(* IEC 61131-3 sources: scada_scout/plc_programs (part 4) *)

(* ---- PRG_GPS02LBB01.st ---- *)
(* ========================================================================
   PLC PROGRAM: PRG_GPS02LBB01
   IED: GPS02LBB01
   Device: GPS02LBB01
   Generated: 2026-02-05 10:51:36

   This program runs cyclically (default 100ms) and has access to all
   data points of the associated IEC 61850 device. Users can add custom
   logic in the designated sections below.
   ======================================================================== *)

PROGRAM PRG_GPS02LBB01
VAR
    (* ====== System Variables ====== *)
    cycle_count: UDINT := 0;           (* Increments each scan cycle *)
    first_scan: BOOL := TRUE;          (* TRUE only on first execution *)
    scan_time_ms: REAL := 0.0;         (* Last scan time in milliseconds *)

    (* ====== IED Connection Status ====== *)
    ied_connected: BOOL := FALSE;      (* TRUE when IED server is running *)
    ied_name: STRING := 'GPS02LBB01';
    device_name: STRING := 'GPS02LBB01';

    (* ====== Logical Devices ====== *)
    (* Available LDs: AnUn_ArcProtInput1, Application, BinIO, BinIO_BinaryInputs, BinIO_BinaryOutputs, CB1, CB1_Fundamental, Ds1, Ds2, Mod1, Mod1_Channel1, Mod2, Mod2_Channel1, Mod3, Mod3_Channel1, PowS, PowS_MeasPointI3ph1, PowS_MeasPointV3ph1, Rec, Rec_FaultRecorder, VI3p1, VI3p1_5051NOCgndB1, VI3p1_5051OC3phase1, VI3p1_67DirOC3phB1, VI3p1_67NDirOCgndB1, VI3p1_ArcProtection1, VI3p1_Energy, VI3p1_FundSymComp, VI3p1_OperationalValues, VI3p1_ProcessMonitor, VI3p1_ExternalTrip1, VI3p1_ExternalTrip2, VI3p1_ExternalTrip3, ComSupervision, ComSupervision_GOOSE *)

    (* ====== User Variables ====== *)
    (* Add your custom variables here *)
    (* Example:
    timer1: TON;
    counter: INT := 0;
    status_word: WORD;
    *)

END_VAR

(* ======================================================================
   INITIALIZATION SECTION
   Runs once on first scan. Use for setup and initialization.
   ====================================================================== *)
IF first_scan THEN
    (* Initialize user variables here *)
    cycle_count := 0;

    (* Log program start *)
    (* SCADA_LOG('INFO', CONCAT('PLC Program started: ', device_name)); *)

    first_scan := FALSE;
END_IF;

(* ======================================================================
   MAIN CYCLIC EXECUTION
   This section runs continuously every scan cycle (default 100ms).
   ====================================================================== *)

(* Increment cycle counter *)
cycle_count := cycle_count + 1;

(* ====== USER LOGIC SECTION 1: Pre-Processing ====== *)
(* Add logic that should run before main processing *)
(* Example:
IF ied_connected THEN
    (* Read IED data points *)
    (* status_word := READ_IED_DATA(device_name, 'LD0/MMXU1$MX$TotW$mag'); *)
END_IF;
*)

(* ====== USER LOGIC SECTION 2: Main Processing ====== *)
(* Add your main control logic here *)
(* Example:
IF counter > 100 THEN
    counter := 0;
    (* Perform periodic action *)
END_IF;
counter := counter + 1;
*)

(* ====== USER LOGIC SECTION 3: Post-Processing ====== *)
(* Add logic for outputs, writes, and cleanup *)
(* Example:
IF ied_connected THEN
    (* Write control commands to IED *)
    (* WRITE_IED_CONTROL(device_name, 'LD0/CSWI1$CO$Pos', TRUE); *)
END_IF;
*)

(* ====== Built-in Functions Available ====== *)
(*
   READ_IED_DATA(device: STRING, ref: STRING): ANY
       - Read data from IED object reference
       - Example: READ_IED_DATA('MyIED', 'LD0/MMXU1$MX$TotW$mag')

   WRITE_IED_DATA(device: STRING, ref: STRING, value: ANY): BOOL
       - Write data to IED object reference
       - Returns TRUE on success

   WRITE_IED_CONTROL(device: STRING, ref: STRING, value: ANY): BOOL
       - Send control command to IED
       - Returns TRUE on success

   SCADA_LOG(level: STRING, message: STRING)
       - Log message to event log
       - Levels: 'INFO', 'WARNING', 'ERROR'

   GET_DEVICE_STATUS(device: STRING): BOOL
       - Check if device is connected
*)

END_PROGRAM

(* ---- PRG_GPS02MCB01.st ---- *)
(* ========================================================================
   PLC PROGRAM: PRG_GPS02MCB01
   IED: GPS02MCB01
   Device: GPS02MCB01
   Generated: 2026-02-05 10:51:25

   This program runs cyclically (default 100ms) and has access to all
   data points of the associated IEC 61850 device. Users can add custom
   logic in the designated sections below.
   ======================================================================== *)

PROGRAM PRG_GPS02MCB01
VAR
    (* ====== System Variables ====== *)
    cycle_count: UDINT := 0;           (* Increments each scan cycle *)
    first_scan: BOOL := TRUE;          (* TRUE only on first execution *)
    scan_time_ms: REAL := 0.0;         (* Last scan time in milliseconds *)

    (* ====== IED Connection Status ====== *)
    ied_connected: BOOL := FALSE;      (* TRUE when IED server is running *)
    ied_name: STRING := 'GPS02MCB01';
    device_name: STRING := 'GPS02MCB01';

    (* ====== Logical Devices ====== *)
    (* Available LDs: AnUn_ArcProtInput1, Application, BinIO, BinIO_BinaryInputs, BinIO_BinaryOutputs, CB1, CB1_Fundamental, Ds1, Ds2, Mod1, Mod1_Channel1, Mod2, Mod2_Channel1, Mod3, Mod3_Channel1, PowS, PowS_MeasPointI3ph1, PowS_MeasPointV1ph1, PowS_MeasPointV3ph1, Rec, Rec_FaultRecorder, VI1p1, VI1p1_Fundamental, VI3p1, VI3p1_5051NOCgndB1, VI3p1_5051OC3phase1, VI3p1_67DirOC3phB1, VI3p1_67NDirOCgndB1, VI3p1_ArcProtection1, VI3p1_Energy, VI3p1_FundSymComp, VI3p1_OperationalValues, VI3p1_ProcessMonitor, VI3p1_ExternalTrip1, VI3p1_ExternalTrip2, VI3p1_ExternalTrip3, ComSupervision, ComSupervision_GOOSE *)

    (* ====== User Variables ====== *)
    (* Add your custom variables here *)
    (* Example:
    timer1: TON;
    counter: INT := 0;
    status_word: WORD;
    *)

END_VAR

(* ======================================================================
   INITIALIZATION SECTION
   Runs once on first scan. Use for setup and initialization.
   ====================================================================== *)
IF first_scan THEN
    (* Initialize user variables here *)
    cycle_count := 0;

    (* Log program start *)
    (* SCADA_LOG('INFO', CONCAT('PLC Program started: ', device_name)); *)

    first_scan := FALSE;
END_IF;

(* ======================================================================
   MAIN CYCLIC EXECUTION
   This section runs continuously every scan cycle (default 100ms).
   ====================================================================== *)

(* Increment cycle counter *)
cycle_count := cycle_count + 1;

(* ====== USER LOGIC SECTION 1: Pre-Processing ====== *)
(* Add logic that should run before main processing *)
(* Example:
IF ied_connected THEN
    (* Read IED data points *)
    (* status_word := READ_IED_DATA(device_name, 'LD0/MMXU1$MX$TotW$mag'); *)
END_IF;
*)

(* ====== USER LOGIC SECTION 2: Main Processing ====== *)
(* Add your main control logic here *)
(* Example:
IF counter > 100 THEN
    counter := 0;
    (* Perform periodic action *)
END_IF;
counter := counter + 1;
*)

(* ====== USER LOGIC SECTION 3: Post-Processing ====== *)
(* Add logic for outputs, writes, and cleanup *)
(* Example:
IF ied_connected THEN
    (* Write control commands to IED *)
    (* WRITE_IED_CONTROL(device_name, 'LD0/CSWI1$CO$Pos', TRUE); *)
END_IF;
*)

(* ====== Built-in Functions Available ====== *)
(*
   READ_IED_DATA(device: STRING, ref: STRING): ANY
       - Read data from IED object reference
       - Example: READ_IED_DATA('MyIED', 'LD0/MMXU1$MX$TotW$mag')

   WRITE_IED_DATA(device: STRING, ref: STRING, value: ANY): BOOL
       - Write data to IED object reference
       - Returns TRUE on success

   WRITE_IED_CONTROL(device: STRING, ref: STRING, value: ANY): BOOL
       - Send control command to IED
       - Returns TRUE on success

   SCADA_LOG(level: STRING, message: STRING)
       - Log message to event log
       - Levels: 'INFO', 'WARNING', 'ERROR'

   GET_DEVICE_STATUS(device: STRING): BOOL
       - Check if device is connected
*)

END_PROGRAM

(* ---- PRG_GPS03ECB01.st ---- *)
(* ========================================================================
   PLC PROGRAM: PRG_GPS03ECB01
   IED: GPS03ECB01
   Device: GPS03ECB01
   Generated: 2026-02-05 10:52:32

   This program runs cyclically (default 100ms) and has access to all
   data points of the associated IEC 61850 device. Users can add custom
   logic in the designated sections below.
   ======================================================================== *)

PROGRAM PRG_GPS03ECB01
VAR
    (* ====== System Variables ====== *)
    cycle_count: UDINT := 0;           (* Increments each scan cycle *)
    first_scan: BOOL := TRUE;          (* TRUE only on first execution *)
    scan_time_ms: REAL := 0.0;         (* Last scan time in milliseconds *)

    (* ====== IED Connection Status ====== *)
    ied_connected: BOOL := FALSE;      (* TRUE when IED server is running *)
    ied_name: STRING := 'GPS03ECB01';
    device_name: STRING := 'GPS03ECB01';

    (* ====== Logical Devices ====== *)
    (* Available LDs: AnUn_ArcProtInput1, Application, BinIO, BinIO_BinaryInputs, BinIO_BinaryOutputs, CB1, CB1_Fundamental, Ds1, Ds2, Mod1, Mod1_Channel1, Mod2, Mod2_Channel1, Mod3, Mod3_Channel1, PowS, PowS_MeasPointI3ph1, PowS_MeasPointV3ph1, Rec, Rec_FaultRecorder, VI3p1, VI3p1_5051NOCgndB1, VI3p1_5051OC3phase1, VI3p1_67DirOC3phB1, VI3p1_67NDirOCgndB1, VI3p1_ArcProtection1, VI3p1_Energy, VI3p1_FundSymComp, VI3p1_OperationalValues, VI3p1_ProcessMonitor, VI3p1_ExternalTrip1, VI3p1_ExternalTrip2, PowS_MeasPointI1ph1, VI1p1, VI1p1_50N51NOC1phB1, VI1p1_Fundamental, ComSupervision, ComSupervision_GOOSE *)

    (* ====== User Variables ====== *)
    (* Add your custom variables here *)
    (* Example:
    timer1: TON;
    counter: INT := 0;
    status_word: WORD;
    *)

END_VAR

(* ======================================================================
   INITIALIZATION SECTION
   Runs once on first scan. Use for setup and initialization.
   ====================================================================== *)
IF first_scan THEN
    (* Initialize user variables here *)
    cycle_count := 0;

    (* Log program start *)
    (* SCADA_LOG('INFO', CONCAT('PLC Program started: ', device_name)); *)

    first_scan := FALSE;
END_IF;

(* ======================================================================
   MAIN CYCLIC EXECUTION
   This section runs continuously every scan cycle (default 100ms).
   ====================================================================== *)

(* Increment cycle counter *)
cycle_count := cycle_count + 1;

(* ====== USER LOGIC SECTION 1: Pre-Processing ====== *)
(* Add logic that should run before main processing *)
(* Example:
IF ied_connected THEN
    (* Read IED data points *)
    (* status_word := READ_IED_DATA(device_name, 'LD0/MMXU1$MX$TotW$mag'); *)
END_IF;
*)

(* ====== USER LOGIC SECTION 2: Main Processing ====== *)
(* Add your main control logic here *)
(* Example:
IF counter > 100 THEN
    counter := 0;
    (* Perform periodic action *)
END_IF;
counter := counter + 1;
*)

(* ====== USER LOGIC SECTION 3: Post-Processing ====== *)
(* Add logic for outputs, writes, and cleanup *)
(* Example:
IF ied_connected THEN
    (* Write control commands to IED *)
    (* WRITE_IED_CONTROL(device_name, 'LD0/CSWI1$CO$Pos', TRUE); *)
END_IF;
*)

(* ====== Built-in Functions Available ====== *)
(*
   READ_IED_DATA(device: STRING, ref: STRING): ANY
       - Read data from IED object reference
       - Example: READ_IED_DATA('MyIED', 'LD0/MMXU1$MX$TotW$mag')

   WRITE_IED_DATA(device: STRING, ref: STRING, value: ANY): BOOL
       - Write data to IED object reference
       - Returns TRUE on success

   WRITE_IED_CONTROL(device: STRING, ref: STRING, value: ANY): BOOL
       - Send control command to IED
       - Returns TRUE on success

   SCADA_LOG(level: STRING, message: STRING)
       - Log message to event log
       - Levels: 'INFO', 'WARNING', 'ERROR'

   GET_DEVICE_STATUS(device: STRING): BOOL
       - Check if device is connected
*)

END_PROGRAM

(* ---- PRG_GPS03FCB01.st ---- *)
(* ========================================================================
   PLC PROGRAM: PRG_GPS03FCB01
   IED: GPS03FCB01
   Device: GPS03FCB01
   Generated: 2026-02-05 10:52:44

   This program runs cyclically (default 100ms) and has access to all
   data points of the associated IEC 61850 device. Users can add custom
   logic in the designated sections below.
   ======================================================================== *)

PROGRAM PRG_GPS03FCB01
VAR
    (* ====== System Variables ====== *)
    cycle_count: UDINT := 0;           (* Increments each scan cycle *)
    first_scan: BOOL := TRUE;          (* TRUE only on first execution *)
    scan_time_ms: REAL := 0.0;         (* Last scan time in milliseconds *)

    (* ====== IED Connection Status ====== *)
    ied_connected: BOOL := FALSE;      (* TRUE when IED server is running *)
    ied_name: STRING := 'GPS03FCB01';
    device_name: STRING := 'GPS03FCB01';

    (* ====== Logical Devices ====== *)
    (* Available LDs: AnUn_ArcProtInput1, Application, BinIO, BinIO_BinaryInputs, BinIO_BinaryOutputs, CB1, CB1_Fundamental, Ds1, Ds2, Mod1, Mod1_Channel1, Mod2, Mod2_Channel1, Mod3, Mod3_Channel1, PowS, PowS_MeasPointI3ph1, PowS_MeasPointV1ph1, PowS_MeasPointV3ph1, Rec, Rec_FaultRecorder, VI1p1, VI1p1_Fundamental, VI3p1, VI3p1_5051NOCgndB1, VI3p1_5051OC3phase1, VI3p1_67DirOC3phB1, VI3p1_67NDirOCgndB1, VI3p1_ArcProtection1, VI3p1_Energy, VI3p1_FundSymComp, VI3p1_OperationalValues, VI3p1_ProcessMonitor, VI3p1_ExternalTrip1, VI3p1_ExternalTrip2, ComSupervision, ComSupervision_GOOSE *)

    (* ====== User Variables ====== *)
    (* Add your custom variables here *)
    (* Example:
    timer1: TON;
    counter: INT := 0;
    status_word: WORD;
    *)

END_VAR

(* ======================================================================
   INITIALIZATION SECTION
   Runs once on first scan. Use for setup and initialization.
   ====================================================================== *)
IF first_scan THEN
    (* Initialize user variables here *)
    cycle_count := 0;

    (* Log program start *)
    (* SCADA_LOG('INFO', CONCAT('PLC Program started: ', device_name)); *)

    first_scan := FALSE;
END_IF;

(* ======================================================================
   MAIN CYCLIC EXECUTION
   This section runs continuously every scan cycle (default 100ms).
   ====================================================================== *)

(* Increment cycle counter *)
cycle_count := cycle_count + 1;

(* ====== USER LOGIC SECTION 1: Pre-Processing ====== *)
(* Add logic that should run before main processing *)
(* Example:
IF ied_connected THEN
    (* Read IED data points *)
    (* status_word := READ_IED_DATA(device_name, 'LD0/MMXU1$MX$TotW$mag'); *)
END_IF;
*)

(* ====== USER LOGIC SECTION 2: Main Processing ====== *)
(* Add your main control logic here *)
(* Example:
IF counter > 100 THEN
    counter := 0;
    (* Perform periodic action *)
END_IF;
counter := counter + 1;
*)

(* ====== USER LOGIC SECTION 3: Post-Processing ====== *)
(* Add logic for outputs, writes, and cleanup *)
(* Example:
IF ied_connected THEN
    (* Write control commands to IED *)
    (* WRITE_IED_CONTROL(device_name, 'LD0/CSWI1$CO$Pos', TRUE); *)
END_IF;
*)

(* ====== Built-in Functions Available ====== *)
(*
   READ_IED_DATA(device: STRING, ref: STRING): ANY
       - Read data from IED object reference
       - Example: READ_IED_DATA('MyIED', 'LD0/MMXU1$MX$TotW$mag')

   WRITE_IED_DATA(device: STRING, ref: STRING, value: ANY): BOOL
       - Write data to IED object reference
       - Returns TRUE on success

   WRITE_IED_CONTROL(device: STRING, ref: STRING, value: ANY): BOOL
       - Send control command to IED
       - Returns TRUE on success

   SCADA_LOG(level: STRING, message: STRING)
       - Log message to event log
       - Levels: 'INFO', 'WARNING', 'ERROR'

   GET_DEVICE_STATUS(device: STRING): BOOL
       - Check if device is connected
*)

END_PROGRAM

(* ---- PRG_GPS03FCB02.st ---- *)
(* ========================================================================
   PLC PROGRAM: PRG_GPS03FCB02
   IED: GPS03FCB02
   Device: GPS03FCB02
   Generated: 2026-02-05 10:52:42

   This program runs cyclically (default 100ms) and has access to all
   data points of the associated IEC 61850 device. Users can add custom
   logic in the designated sections below.
   ======================================================================== *)

PROGRAM PRG_GPS03FCB02
VAR
    (* ====== System Variables ====== *)
    cycle_count: UDINT := 0;           (* Increments each scan cycle *)
    first_scan: BOOL := TRUE;          (* TRUE only on first execution *)
    scan_time_ms: REAL := 0.0;         (* Last scan time in milliseconds *)

    (* ====== IED Connection Status ====== *)
    ied_connected: BOOL := FALSE;      (* TRUE when IED server is running *)
    ied_name: STRING := 'GPS03FCB02';
    device_name: STRING := 'GPS03FCB02';

    (* ====== Logical Devices ====== *)
    (* Available LDs: AnUn_ArcProtInput1, Application, BinIO, BinIO_BinaryInputs, BinIO_BinaryOutputs, CB1, CB1_Fundamental, Ds1, Ds2, Mod1, Mod1_Channel1, Mod2, Mod2_Channel1, Mod3, Mod3_Channel1, PowS, PowS_MeasPointI3ph1, PowS_MeasPointV1ph1, PowS_MeasPointV3ph1, Rec, Rec_FaultRecorder, VI1p1, VI1p1_Fundamental, VI3p1, VI3p1_5051NOCgndB1, VI3p1_5051OC3phase1, VI3p1_67DirOC3phB1, VI3p1_67NDirOCgndB1, VI3p1_ArcProtection1, VI3p1_Energy, VI3p1_FundSymComp, VI3p1_OperationalValues, VI3p1_ProcessMonitor, VI3p1_ExternalTrip1, VI3p1_ExternalTrip2, ComSupervision, ComSupervision_GOOSE *)

    (* ====== User Variables ====== *)
    (* Add your custom variables here *)
    (* Example:
    timer1: TON;
    counter: INT := 0;
    status_word: WORD;
    *)

END_VAR

(* ======================================================================
   INITIALIZATION SECTION
   Runs once on first scan. Use for setup and initialization.
   ====================================================================== *)
IF first_scan THEN
    (* Initialize user variables here *)
    cycle_count := 0;

    (* Log program start *)
    (* SCADA_LOG('INFO', CONCAT('PLC Program started: ', device_name)); *)

    first_scan := FALSE;
END_IF;

(* ======================================================================
   MAIN CYCLIC EXECUTION
   This section runs continuously every scan cycle (default 100ms).
   ====================================================================== *)

(* Increment cycle counter *)
cycle_count := cycle_count + 1;

(* ====== USER LOGIC SECTION 1: Pre-Processing ====== *)
(* Add logic that should run before main processing *)
(* Example:
IF ied_connected THEN
    (* Read IED data points *)
    (* status_word := READ_IED_DATA(device_name, 'LD0/MMXU1$MX$TotW$mag'); *)
END_IF;
*)

(* ====== USER LOGIC SECTION 2: Main Processing ====== *)
(* Add your main control logic here *)
(* Example:
IF counter > 100 THEN
    counter := 0;
    (* Perform periodic action *)
END_IF;
counter := counter + 1;
*)

(* ====== USER LOGIC SECTION 3: Post-Processing ====== *)
(* Add logic for outputs, writes, and cleanup *)
(* Example:
IF ied_connected THEN
    (* Write control commands to IED *)
    (* WRITE_IED_CONTROL(device_name, 'LD0/CSWI1$CO$Pos', TRUE); *)
END_IF;
*)

(* ====== Built-in Functions Available ====== *)
(*
   READ_IED_DATA(device: STRING, ref: STRING): ANY
       - Read data from IED object reference
       - Example: READ_IED_DATA('MyIED', 'LD0/MMXU1$MX$TotW$mag')

   WRITE_IED_DATA(device: STRING, ref: STRING, value: ANY): BOOL
       - Write data to IED object reference
       - Returns TRUE on success

   WRITE_IED_CONTROL(device: STRING, ref: STRING, value: ANY): BOOL
       - Send control command to IED
       - Returns TRUE on success

   SCADA_LOG(level: STRING, message: STRING)
       - Log message to event log
       - Levels: 'INFO', 'WARNING', 'ERROR'

   GET_DEVICE_STATUS(device: STRING): BOOL
       - Check if device is connected
*)

END_PROGRAM

(* ---- PRG_GPS03FCB03.st ---- *)
(* ========================================================================
   PLC PROGRAM: PRG_GPS03FCB03
   IED: GPS03FCB03
   Device: GPS03FCB03
   Generated: 2026-02-05 10:53:26

   This program runs cyclically (default 100ms) and has access to all
   data points of the associated IEC 61850 device. Users can add custom
   logic in the designated sections below.
   ======================================================================== *)

PROGRAM PRG_GPS03FCB03
VAR
    (* ====== System Variables ====== *)
    cycle_count: UDINT := 0;           (* Increments each scan cycle *)
    first_scan: BOOL := TRUE;          (* TRUE only on first execution *)
    scan_time_ms: REAL := 0.0;         (* Last scan time in milliseconds *)

    (* ====== IED Connection Status ====== *)
    ied_connected: BOOL := FALSE;      (* TRUE when IED server is running *)
    ied_name: STRING := 'GPS03FCB03';
    device_name: STRING := 'GPS03FCB03';

    (* ====== Logical Devices ====== *)
    (* Available LDs: AnUn_ArcProtInput1, Application, BinIO, BinIO_BinaryInputs, BinIO_BinaryOutputs, CB1, CB1_Fundamental, Ds1, Ds2, Mod1, Mod1_Channel1, Mod2, Mod2_Channel1, Mod3, Mod3_Channel1, PowS, PowS_MeasPointI3ph1, PowS_MeasPointV1ph1, PowS_MeasPointV3ph1, Rec, Rec_FaultRecorder, VI1p1, VI1p1_Fundamental, VI3p1, VI3p1_5051NOCgndB1, VI3p1_5051OC3phase1, VI3p1_67DirOC3phB1, VI3p1_67NDirOCgndB1, VI3p1_ArcProtection1, VI3p1_Energy, VI3p1_FundSymComp, VI3p1_OperationalValues, VI3p1_ProcessMonitor, VI3p1_ExternalTrip1, VI3p1_ExternalTrip2, VI3p1_ExternalTrip3, ComSupervision, ComSupervision_GOOSE *)

    (* ====== User Variables ====== *)
    (* Add your custom variables here *)
    (* Example:
    timer1: TON;
    counter: INT := 0;
    status_word: WORD;
    *)

END_VAR

(* ======================================================================
   INITIALIZATION SECTION
   Runs once on first scan. Use for setup and initialization.
   ====================================================================== *)
IF first_scan THEN
    (* Initialize user variables here *)
    cycle_count := 0;

    (* Log program start *)
    (* SCADA_LOG('INFO', CONCAT('PLC Program started: ', device_name)); *)

    first_scan := FALSE;
END_IF;

(* ======================================================================
   MAIN CYCLIC EXECUTION
   This section runs continuously every scan cycle (default 100ms).
   ====================================================================== *)

(* Increment cycle counter *)
cycle_count := cycle_count + 1;

(* ====== USER LOGIC SECTION 1: Pre-Processing ====== *)
(* Add logic that should run before main processing *)
(* Example:
IF ied_connected THEN
    (* Read IED data points *)
    (* status_word := READ_IED_DATA(device_name, 'LD0/MMXU1$MX$TotW$mag'); *)
END_IF;
*)

(* ====== USER LOGIC SECTION 2: Main Processing ====== *)
(* Add your main control logic here *)
(* Example:
IF counter > 100 THEN
    counter := 0;
    (* Perform periodic action *)
END_IF;
counter := counter + 1;
*)

(* ====== USER LOGIC SECTION 3: Post-Processing ====== *)
(* Add logic for outputs, writes, and cleanup *)
(* Example:
IF ied_connected THEN
    (* Write control commands to IED *)
    (* WRITE_IED_CONTROL(device_name, 'LD0/CSWI1$CO$Pos', TRUE); *)
END_IF;
*)

(* ====== Built-in Functions Available ====== *)
(*
   READ_IED_DATA(device: STRING, ref: STRING): ANY
       - Read data from IED object reference
       - Example: READ_IED_DATA('MyIED', 'LD0/MMXU1$MX$TotW$mag')

   WRITE_IED_DATA(device: STRING, ref: STRING, value: ANY): BOOL
       - Write data to IED object reference
       - Returns TRUE on success

   WRITE_IED_CONTROL(device: STRING, ref: STRING, value: ANY): BOOL
       - Send control command to IED
       - Returns TRUE on success

   SCADA_LOG(level: STRING, message: STRING)
       - Log message to event log
       - Levels: 'INFO', 'WARNING', 'ERROR'

   GET_DEVICE_STATUS(device: STRING): BOOL
       - Check if device is connected
*)

END_PROGRAM

(* ---- PRG_GPS03GCB01.st ---- *)
(* ========================================================================
   PLC PROGRAM: PRG_GPS03GCB01
   IED: GPS03GCB01
   Device: GPS03GCB01
   Generated: 2026-02-05 10:53:22

   This program runs cyclically (default 100ms) and has access to all
   data points of the associated IEC 61850 device. Users can add custom
   logic in the designated sections below.
   ======================================================================== *)

PROGRAM PRG_GPS03GCB01
VAR
    (* ====== System Variables ====== *)
    cycle_count: UDINT := 0;           (* Increments each scan cycle *)
    first_scan: BOOL := TRUE;          (* TRUE only on first execution *)
    scan_time_ms: REAL := 0.0;         (* Last scan time in milliseconds *)

    (* ====== IED Connection Status ====== *)
    ied_connected: BOOL := FALSE;      (* TRUE when IED server is running *)
    ied_name: STRING := 'GPS03GCB01';
    device_name: STRING := 'GPS03GCB01';

    (* ====== Logical Devices ====== *)
    (* Available LDs: AnUn_ArcProtInput1, Application, BinIO, BinIO_BinaryInputs, BinIO_BinaryOutputs, CB1, CB1_25Synchronization, CB1_Fundamental, Ds1, Ds2, Mod1, Mod1_Channel1, Mod2, Mod2_Channel1, Mod3, Mod3_Channel1, PowS, PowS_MeasPointI3ph1, PowS_MeasPointV1ph1, PowS_MeasPointV3ph1, Rec, Rec_FaultRecorder, VI1p1, VI1p1_Fundamental, VI3p1, VI3p1_5051NOCgndB1, VI3p1_5051OC3phase1, VI3p1_67DirOC3phB1, VI3p1_67NDirOCgndB1, VI3p1_ArcProtection1, VI3p1_Energy, VI3p1_FundSymComp, VI3p1_OperationalValues, VI3p1_ProcessMonitor, VI3p1_ExternalTrip1, VI3p1_ExternalTrip2, ComSupervision, ComSupervision_GOOSE *)

    (* ====== User Variables ====== *)
    (* Add your custom variables here *)
    (* Example:
    timer1: TON;
    counter: INT := 0;
    status_word: WORD;
    *)

END_VAR

(* ======================================================================
   INITIALIZATION SECTION
   Runs once on first scan. Use for setup and initialization.
   ====================================================================== *)
IF first_scan THEN
    (* Initialize user variables here *)
    cycle_count := 0;

    (* Log program start *)
    (* SCADA_LOG('INFO', CONCAT('PLC Program started: ', device_name)); *)

    first_scan := FALSE;
END_IF;

(* ======================================================================
   MAIN CYCLIC EXECUTION
   This section runs continuously every scan cycle (default 100ms).
   ====================================================================== *)

(* Increment cycle counter *)
cycle_count := cycle_count + 1;

(* ====== USER LOGIC SECTION 1: Pre-Processing ====== *)
(* Add logic that should run before main processing *)
(* Example:
IF ied_connected THEN
    (* Read IED data points *)
    (* status_word := READ_IED_DATA(device_name, 'LD0/MMXU1$MX$TotW$mag'); *)
END_IF;
*)

(* ====== USER LOGIC SECTION 2: Main Processing ====== *)
(* Add your main control logic here *)
(* Example:
IF counter > 100 THEN
    counter := 0;
    (* Perform periodic action *)
END_IF;
counter := counter + 1;
*)

(* ====== USER LOGIC SECTION 3: Post-Processing ====== *)
(* Add logic for outputs, writes, and cleanup *)
(* Example:
IF ied_connected THEN
    (* Write control commands to IED *)
    (* WRITE_IED_CONTROL(device_name, 'LD0/CSWI1$CO$Pos', TRUE); *)
END_IF;
*)

(* ====== Built-in Functions Available ====== *)
(*
   READ_IED_DATA(device: STRING, ref: STRING): ANY
       - Read data from IED object reference
       - Example: READ_IED_DATA('MyIED', 'LD0/MMXU1$MX$TotW$mag')

   WRITE_IED_DATA(device: STRING, ref: STRING, value: ANY): BOOL
       - Write data to IED object reference
       - Returns TRUE on success

   WRITE_IED_CONTROL(device: STRING, ref: STRING, value: ANY): BOOL
       - Send control command to IED
       - Returns TRUE on success

   SCADA_LOG(level: STRING, message: STRING)
       - Log message to event log
       - Levels: 'INFO', 'WARNING', 'ERROR'

   GET_DEVICE_STATUS(device: STRING): BOOL
       - Check if device is connected
*)

END_PROGRAM

(* ---- PRG_GPS03GCB02.st ---- *)
(* ========================================================================
   PLC PROGRAM: PRG_GPS03GCB02
   IED: GPS03GCB02
   Device: GPS03GCB02
   Generated: 2026-02-05 10:53:14

   This program runs cyclically (default 100ms) and has access to all
   data points of the associated IEC 61850 device. Users can add custom
   logic in the designated sections below.
   ======================================================================== *)

PROGRAM PRG_GPS03GCB02
VAR
    (* ====== System Variables ====== *)
    cycle_count: UDINT := 0;           (* Increments each scan cycle *)
    first_scan: BOOL := TRUE;          (* TRUE only on first execution *)
    scan_time_ms: REAL := 0.0;         (* Last scan time in milliseconds *)

    (* ====== IED Connection Status ====== *)
    ied_connected: BOOL := FALSE;      (* TRUE when IED server is running *)
    ied_name: STRING := 'GPS03GCB02';
    device_name: STRING := 'GPS03GCB02';

    (* ====== Logical Devices ====== *)
    (* Available LDs: AnUn_ArcProtInput1, Application, BinIO, BinIO_BinaryInputs, BinIO_BinaryOutputs, CB1, CB1_25Synchronization, CB1_Fundamental, Ds1, Ds2, Mod1, Mod1_Channel1, Mod2, Mod2_Channel1, Mod3, Mod3_Channel1, PowS, PowS_MeasPointI3ph1, PowS_MeasPointV1ph1, PowS_MeasPointV3ph1, Rec, Rec_FaultRecorder, VI1p1, VI1p1_Fundamental, VI3p1, VI3p1_5051NOCgndB1, VI3p1_5051OC3phase1, VI3p1_67DirOC3phB1, VI3p1_67NDirOCgndB1, VI3p1_ArcProtection1, VI3p1_Energy, VI3p1_FundSymComp, VI3p1_OperationalValues, VI3p1_ProcessMonitor, VI3p1_ExternalTrip1, VI3p1_ExternalTrip2, ComSupervision, ComSupervision_GOOSE *)

    (* ====== User Variables ====== *)
    (* Add your custom variables here *)
    (* Example:
    timer1: TON;
    counter: INT := 0;
    status_word: WORD;
    *)

END_VAR

(* ======================================================================
   INITIALIZATION SECTION
   Runs once on first scan. Use for setup and initialization.
   ====================================================================== *)
IF first_scan THEN
    (* Initialize user variables here *)
    cycle_count := 0;

    (* Log program start *)
    (* SCADA_LOG('INFO', CONCAT('PLC Program started: ', device_name)); *)

    first_scan := FALSE;
END_IF;

(* ======================================================================
   MAIN CYCLIC EXECUTION
   This section runs continuously every scan cycle (default 100ms).
   ====================================================================== *)

(* Increment cycle counter *)
cycle_count := cycle_count + 1;

(* ====== USER LOGIC SECTION 1: Pre-Processing ====== *)
(* Add logic that should run before main processing *)
(* Example:
IF ied_connected THEN
    (* Read IED data points *)
    (* status_word := READ_IED_DATA(device_name, 'LD0/MMXU1$MX$TotW$mag'); *)
END_IF;
*)

(* ====== USER LOGIC SECTION 2: Main Processing ====== *)
(* Add your main control logic here *)
(* Example:
IF counter > 100 THEN
    counter := 0;
    (* Perform periodic action *)
END_IF;
counter := counter + 1;
*)

(* ====== USER LOGIC SECTION 3: Post-Processing ====== *)
(* Add logic for outputs, writes, and cleanup *)
(* Example:
IF ied_connected THEN
    (* Write control commands to IED *)
    (* WRITE_IED_CONTROL(device_name, 'LD0/CSWI1$CO$Pos', TRUE); *)
END_IF;
*)

(* ====== Built-in Functions Available ====== *)
(*
   READ_IED_DATA(device: STRING, ref: STRING): ANY
       - Read data from IED object reference
       - Example: READ_IED_DATA('MyIED', 'LD0/MMXU1$MX$TotW$mag')

   WRITE_IED_DATA(device: STRING, ref: STRING, value: ANY): BOOL
       - Write data to IED object reference
       - Returns TRUE on success

   WRITE_IED_CONTROL(device: STRING, ref: STRING, value: ANY): BOOL
       - Send control command to IED
       - Returns TRUE on success

   SCADA_LOG(level: STRING, message: STRING)
       - Log message to event log
       - Levels: 'INFO', 'WARNING', 'ERROR'

   GET_DEVICE_STATUS(device: STRING): BOOL
       - Check if device is connected
*)

END_PROGRAM

(* ---- PRG_GPS03GCB03.st ---- *)
(* ========================================================================
   PLC PROGRAM: PRG_GPS03GCB03
   IED: GPS03GCB03
   Device: GPS03GCB03
   Generated: 2026-02-05 10:53:06

   This program runs cyclically (default 100ms) and has access to all
   data points of the associated IEC 61850 device. Users can add custom
   logic in the designated sections below.
   ======================================================================== *)

PROGRAM PRG_GPS03GCB03
VAR
    (* ====== System Variables ====== *)
    cycle_count: UDINT := 0;           (* Increments each scan cycle *)
    first_scan: BOOL := TRUE;          (* TRUE only on first execution *)
    scan_time_ms: REAL := 0.0;         (* Last scan time in milliseconds *)

    (* ====== IED Connection Status ====== *)
    ied_connected: BOOL := FALSE;      (* TRUE when IED server is running *)
    ied_name: STRING := 'GPS03GCB03';
    device_name: STRING := 'GPS03GCB03';

    (* ====== Logical Devices ====== *)
    (* Available LDs: AnUn_ArcProtInput1, Application, BinIO, BinIO_BinaryInputs, BinIO_BinaryOutputs, CB1, CB1_25Synchronization, CB1_Fundamental, Ds1, Ds2, Mod1, Mod1_Channel1, Mod2, Mod2_Channel1, Mod3, Mod3_Channel1, PowS, PowS_MeasPointI3ph1, PowS_MeasPointV1ph1, PowS_MeasPointV3ph1, Rec, Rec_FaultRecorder, VI1p1, VI1p1_Fundamental, VI3p1, VI3p1_5051NOCgndB1, VI3p1_5051OC3phase1, VI3p1_67DirOC3phB1, VI3p1_67NDirOCgndB1, VI3p1_ArcProtection1, VI3p1_Energy, VI3p1_FundSymComp, VI3p1_OperationalValues, VI3p1_ProcessMonitor, VI3p1_ExternalTrip1, VI3p1_ExternalTrip2, ComSupervision, ComSupervision_GOOSE *)

    (* ====== User Variables ====== *)
    (* Add your custom variables here *)
    (* Example:
    timer1: TON;
    counter: INT := 0;
    status_word: WORD;
    *)

END_VAR

(* ======================================================================
   INITIALIZATION SECTION
   Runs once on first scan. Use for setup and initialization.
   ====================================================================== *)
IF first_scan THEN
    (* Initialize user variables here *)
    cycle_count := 0;

    (* Log program start *)
    (* SCADA_LOG('INFO', CONCAT('PLC Program started: ', device_name)); *)

    first_scan := FALSE;
END_IF;

(* ======================================================================
   MAIN CYCLIC EXECUTION
   This section runs continuously every scan cycle (default 100ms).
   ====================================================================== *)

(* Increment cycle counter *)
cycle_count := cycle_count + 1;

(* ====== USER LOGIC SECTION 1: Pre-Processing ====== *)
(* Add logic that should run before main processing *)
(* Example:
IF ied_connected THEN
    (* Read IED data points *)
    (* status_word := READ_IED_DATA(device_name, 'LD0/MMXU1$MX$TotW$mag'); *)
END_IF;
*)

(* ====== USER LOGIC SECTION 2: Main Processing ====== *)
(* Add your main control logic here *)
(* Example:
IF counter > 100 THEN
    counter := 0;
    (* Perform periodic action *)
END_IF;
counter := counter + 1;
*)

(* ====== USER LOGIC SECTION 3: Post-Processing ====== *)
(* Add logic for outputs, writes, and cleanup *)
(* Example:
IF ied_connected THEN
    (* Write control commands to IED *)
    (* WRITE_IED_CONTROL(device_name, 'LD0/CSWI1$CO$Pos', TRUE); *)
END_IF;
*)

(* ====== Built-in Functions Available ====== *)
(*
   READ_IED_DATA(device: STRING, ref: STRING): ANY
       - Read data from IED object reference
       - Example: READ_IED_DATA('MyIED', 'LD0/MMXU1$MX$TotW$mag')

   WRITE_IED_DATA(device: STRING, ref: STRING, value: ANY): BOOL
       - Write data to IED object reference
       - Returns TRUE on success

   WRITE_IED_CONTROL(device: STRING, ref: STRING, value: ANY): BOOL
       - Send control command to IED
       - Returns TRUE on success

   SCADA_LOG(level: STRING, message: STRING)
       - Log message to event log
       - Levels: 'INFO', 'WARNING', 'ERROR'

   GET_DEVICE_STATUS(device: STRING): BOOL
       - Check if device is connected
*)

END_PROGRAM

(* ---- PRG_GPS03GCB04.st ---- *)
(* ========================================================================
   PLC PROGRAM: PRG_GPS03GCB04
   IED: GPS03GCB04
   Device: GPS03GCB04
   Generated: 2026-02-05 10:53:00

   This program runs cyclically (default 100ms) and has access to all
   data points of the associated IEC 61850 device. Users can add custom
   logic in the designated sections below.
   ======================================================================== *)

PROGRAM PRG_GPS03GCB04
VAR
    (* ====== System Variables ====== *)
    cycle_count: UDINT := 0;           (* Increments each scan cycle *)
    first_scan: BOOL := TRUE;          (* TRUE only on first execution *)
    scan_time_ms: REAL := 0.0;         (* Last scan time in milliseconds *)

    (* ====== IED Connection Status ====== *)
    ied_connected: BOOL := FALSE;      (* TRUE when IED server is running *)
    ied_name: STRING := 'GPS03GCB04';
    device_name: STRING := 'GPS03GCB04';

    (* ====== Logical Devices ====== *)
    (* Available LDs: AnUn_ArcProtInput1, Application, BinIO, BinIO_BinaryInputs, BinIO_BinaryOutputs, CB1, CB1_25Synchronization, CB1_Fundamental, Ds1, Ds2, Mod1, Mod1_Channel1, Mod2, Mod2_Channel1, Mod3, Mod3_Channel1, PowS, PowS_MeasPointI3ph1, PowS_MeasPointV1ph1, PowS_MeasPointV3ph1, Rec, Rec_FaultRecorder, VI1p1, VI1p1_Fundamental, VI3p1, VI3p1_5051NOCgndB1, VI3p1_5051OC3phase1, VI3p1_67DirOC3phB1, VI3p1_67NDirOCgndB1, VI3p1_ArcProtection1, VI3p1_Energy, VI3p1_FundSymComp, VI3p1_OperationalValues, VI3p1_ProcessMonitor, VI3p1_ExternalTrip1, VI3p1_ExternalTrip2, ComSupervision, ComSupervision_GOOSE *)

    (* ====== User Variables ====== *)
    (* Add your custom variables here *)
    (* Example:
    timer1: TON;
    counter: INT := 0;
    status_word: WORD;
    *)

END_VAR

(* ======================================================================
   INITIALIZATION SECTION
   Runs once on first scan. Use for setup and initialization.
   ====================================================================== *)
IF first_scan THEN
    (* Initialize user variables here *)
    cycle_count := 0;

    (* Log program start *)
    (* SCADA_LOG('INFO', CONCAT('PLC Program started: ', device_name)); *)

    first_scan := FALSE;
END_IF;

(* ======================================================================
   MAIN CYCLIC EXECUTION
   This section runs continuously every scan cycle (default 100ms).
   ====================================================================== *)

(* Increment cycle counter *)
cycle_count := cycle_count + 1;

(* ====== USER LOGIC SECTION 1: Pre-Processing ====== *)
(* Add logic that should run before main processing *)
(* Example:
IF ied_connected THEN
    (* Read IED data points *)
    (* status_word := READ_IED_DATA(device_name, 'LD0/MMXU1$MX$TotW$mag'); *)
END_IF;
*)

(* ====== USER LOGIC SECTION 2: Main Processing ====== *)
(* Add your main control logic here *)
(* Example:
IF counter > 100 THEN
    counter := 0;
    (* Perform periodic action *)
END_IF;
counter := counter + 1;
*)

(* ====== USER LOGIC SECTION 3: Post-Processing ====== *)
(* Add logic for outputs, writes, and cleanup *)
(* Example:
IF ied_connected THEN
    (* Write control commands to IED *)
    (* WRITE_IED_CONTROL(device_name, 'LD0/CSWI1$CO$Pos', TRUE); *)
END_IF;
*)

(* ====== Built-in Functions Available ====== *)
(*
   READ_IED_DATA(device: STRING, ref: STRING): ANY
       - Read data from IED object reference
       - Example: READ_IED_DATA('MyIED', 'LD0/MMXU1$MX$TotW$mag')

   WRITE_IED_DATA(device: STRING, ref: STRING, value: ANY): BOOL
       - Write data to IED object reference
       - Returns TRUE on success

   WRITE_IED_CONTROL(device: STRING, ref: STRING, value: ANY): BOOL
       - Send control command to IED
       - Returns TRUE on success

   SCADA_LOG(level: STRING, message: STRING)
       - Log message to event log
       - Levels: 'INFO', 'WARNING', 'ERROR'

   GET_DEVICE_STATUS(device: STRING): BOOL
       - Check if device is connected
*)

END_PROGRAM

(* ---- PRG_GPS03GCB05.st ---- *)
(* ========================================================================
   PLC PROGRAM: PRG_GPS03GCB05
   IED: GPS03GCB05
   Device: GPS03GCB05
   Generated: 2026-02-05 10:52:56

   This program runs cyclically (default 100ms) and has access to all
   data points of the associated IEC 61850 device. Users can add custom
   logic in the designated sections below.
   ======================================================================== *)

PROGRAM PRG_GPS03GCB05
VAR
    (* ====== System Variables ====== *)
    cycle_count: UDINT := 0;           (* Increments each scan cycle *)
    first_scan: BOOL := TRUE;          (* TRUE only on first execution *)
    scan_time_ms: REAL := 0.0;         (* Last scan time in milliseconds *)

    (* ====== IED Connection Status ====== *)
    ied_connected: BOOL := FALSE;      (* TRUE when IED server is running *)
    ied_name: STRING := 'GPS03GCB05';
    device_name: STRING := 'GPS03GCB05';

    (* ====== Logical Devices ====== *)
    (* Available LDs: AnUn_ArcProtInput1, Application, BinIO, BinIO_BinaryInputs, BinIO_BinaryOutputs, CB1, CB1_25Synchronization, CB1_Fundamental, Ds1, Ds2, Mod1, Mod1_Channel1, Mod2, Mod2_Channel1, Mod3, Mod3_Channel1, PowS, PowS_MeasPointI3ph1, PowS_MeasPointV1ph1, PowS_MeasPointV3ph1, Rec, Rec_FaultRecorder, VI1p1, VI1p1_Fundamental, VI3p1, VI3p1_5051NOCgndB1, VI3p1_5051OC3phase1, VI3p1_67DirOC3phB1, VI3p1_67NDirOCgndB1, VI3p1_ArcProtection1, VI3p1_Energy, VI3p1_FundSymComp, VI3p1_OperationalValues, VI3p1_ProcessMonitor, VI3p1_ExternalTrip1, VI3p1_ExternalTrip2, ComSupervision, ComSupervision_GOOSE *)

    (* ====== User Variables ====== *)
    (* Add your custom variables here *)
    (* Example:
    timer1: TON;
    counter: INT := 0;
    status_word: WORD;
    *)

END_VAR

(* ======================================================================
   INITIALIZATION SECTION
   Runs once on first scan. Use for setup and initialization.
   ====================================================================== *)
IF first_scan THEN
    (* Initialize user variables here *)
    cycle_count := 0;

    (* Log program start *)
    (* SCADA_LOG('INFO', CONCAT('PLC Program started: ', device_name)); *)

    first_scan := FALSE;
END_IF;

(* ======================================================================
   MAIN CYCLIC EXECUTION
   This section runs continuously every scan cycle (default 100ms).
   ====================================================================== *)

(* Increment cycle counter *)
cycle_count := cycle_count + 1;

(* ====== USER LOGIC SECTION 1: Pre-Processing ====== *)
(* Add logic that should run before main processing *)
(* Example:
IF ied_connected THEN
    (* Read IED data points *)
    (* status_word := READ_IED_DATA(device_name, 'LD0/MMXU1$MX$TotW$mag'); *)
END_IF;
*)

(* ====== USER LOGIC SECTION 2: Main Processing ====== *)
(* Add your main control logic here *)
(* Example:
IF counter > 100 THEN
    counter := 0;
    (* Perform periodic action *)
END_IF;
counter := counter + 1;
*)

(* ====== USER LOGIC SECTION 3: Post-Processing ====== *)
(* Add logic for outputs, writes, and cleanup *)
(* Example:
IF ied_connected THEN
    (* Write control commands to IED *)
    (* WRITE_IED_CONTROL(device_name, 'LD0/CSWI1$CO$Pos', TRUE); *)
END_IF;
*)

(* ====== Built-in Functions Available ====== *)
(*
   READ_IED_DATA(device: STRING, ref: STRING): ANY
       - Read data from IED object reference
       - Example: READ_IED_DATA('MyIED', 'LD0/MMXU1$MX$TotW$mag')

   WRITE_IED_DATA(device: STRING, ref: STRING, value: ANY): BOOL
       - Write data to IED object reference
       - Returns TRUE on success

   WRITE_IED_CONTROL(device: STRING, ref: STRING, value: ANY): BOOL
       - Send control command to IED
       - Returns TRUE on success

   SCADA_LOG(level: STRING, message: STRING)
       - Log message to event log
       - Levels: 'INFO', 'WARNING', 'ERROR'

   GET_DEVICE_STATUS(device: STRING): BOOL
       - Check if device is connected
*)

END_PROGRAM

(* ---- PRG_GPS03GCB06.st ---- *)
(* ========================================================================
   PLC PROGRAM: PRG_GPS03GCB06
   IED: GPS03GCB06
   Device: GPS03GCB06
   Generated: 2026-02-05 10:52:47

   This program runs cyclically (default 100ms) and has access to all
   data points of the associated IEC 61850 device. Users can add custom
   logic in the designated sections below.
   ======================================================================== *)

PROGRAM PRG_GPS03GCB06
VAR
    (* ====== System Variables ====== *)
    cycle_count: UDINT := 0;           (* Increments each scan cycle *)
    first_scan: BOOL := TRUE;          (* TRUE only on first execution *)
    scan_time_ms: REAL := 0.0;         (* Last scan time in milliseconds *)

    (* ====== IED Connection Status ====== *)
    ied_connected: BOOL := FALSE;      (* TRUE when IED server is running *)
    ied_name: STRING := 'GPS03GCB06';
    device_name: STRING := 'GPS03GCB06';

    (* ====== Logical Devices ====== *)
    (* Available LDs: AnUn_ArcProtInput1, Application, BinIO, BinIO_BinaryInputs, BinIO_BinaryOutputs, CB1, CB1_25Synchronization, CB1_Fundamental, Ds1, Ds2, Mod1, Mod1_Channel1, Mod2, Mod2_Channel1, Mod3, Mod3_Channel1, PowS, PowS_MeasPointI3ph1, PowS_MeasPointV1ph1, PowS_MeasPointV3ph1, Rec, Rec_FaultRecorder, VI1p1, VI1p1_Fundamental, VI3p1, VI3p1_5051NOCgndB1, VI3p1_5051OC3phase1, VI3p1_67DirOC3phB1, VI3p1_67NDirOCgndB1, VI3p1_ArcProtection1, VI3p1_Energy, VI3p1_FundSymComp, VI3p1_OperationalValues, VI3p1_ProcessMonitor, VI3p1_ExternalTrip1, VI3p1_ExternalTrip2, ComSupervision, ComSupervision_GOOSE *)

    (* ====== User Variables ====== *)
    (* Add your custom variables here *)
    (* Example:
    timer1: TON;
    counter: INT := 0;
    status_word: WORD;
    *)

END_VAR

(* ======================================================================
   INITIALIZATION SECTION
   Runs once on first scan. Use for setup and initialization.
   ====================================================================== *)
IF first_scan THEN
    (* Initialize user variables here *)
    cycle_count := 0;

    (* Log program start *)
    (* SCADA_LOG('INFO', CONCAT('PLC Program started: ', device_name)); *)

    first_scan := FALSE;
END_IF;

(* ======================================================================
   MAIN CYCLIC EXECUTION
   This section runs continuously every scan cycle (default 100ms).
   ====================================================================== *)

(* Increment cycle counter *)
cycle_count := cycle_count + 1;

(* ====== USER LOGIC SECTION 1: Pre-Processing ====== *)
(* Add logic that should run before main processing *)
(* Example:
IF ied_connected THEN
    (* Read IED data points *)
    (* status_word := READ_IED_DATA(device_name, 'LD0/MMXU1$MX$TotW$mag'); *)
END_IF;
*)

(* ====== USER LOGIC SECTION 2: Main Processing ====== *)
(* Add your main control logic here *)
(* Example:
IF counter > 100 THEN
    counter := 0;
    (* Perform periodic action *)
END_IF;
counter := counter + 1;
*)

(* ====== USER LOGIC SECTION 3: Post-Processing ====== *)
(* Add logic for outputs, writes, and cleanup *)
(* Example:
IF ied_connected THEN
    (* Write control commands to IED *)
    (* WRITE_IED_CONTROL(device_name, 'LD0/CSWI1$CO$Pos', TRUE); *)
END_IF;
*)

(* ====== Built-in Functions Available ====== *)
(*
   READ_IED_DATA(device: STRING, ref: STRING): ANY
       - Read data from IED object reference
       - Example: READ_IED_DATA('MyIED', 'LD0/MMXU1$MX$TotW$mag')

   WRITE_IED_DATA(device: STRING, ref: STRING, value: ANY): BOOL
       - Write data to IED object reference
       - Returns TRUE on success

   WRITE_IED_CONTROL(device: STRING, ref: STRING, value: ANY): BOOL
       - Send control command to IED
       - Returns TRUE on success

   SCADA_LOG(level: STRING, message: STRING)
       - Log message to event log
       - Levels: 'INFO', 'WARNING', 'ERROR'

   GET_DEVICE_STATUS(device: STRING): BOOL
       - Check if device is connected
*)

END_PROGRAM

(* ---- PRG_GPS03GCB07.st ---- *)
(* ========================================================================
   PLC PROGRAM: PRG_GPS03GCB07
   IED: GPS03GCB07
   Device: GPS03GCB07
   Generated: 2026-02-05 10:52:45

   This program runs cyclically (default 100ms) and has access to all
   data points of the associated IEC 61850 device. Users can add custom
   logic in the designated sections below.
   ======================================================================== *)

PROGRAM PRG_GPS03GCB07
VAR
    (* ====== System Variables ====== *)
    cycle_count: UDINT := 0;           (* Increments each scan cycle *)
    first_scan: BOOL := TRUE;          (* TRUE only on first execution *)
    scan_time_ms: REAL := 0.0;         (* Last scan time in milliseconds *)

    (* ====== IED Connection Status ====== *)
    ied_connected: BOOL := FALSE;      (* TRUE when IED server is running *)
    ied_name: STRING := 'GPS03GCB07';
    device_name: STRING := 'GPS03GCB07';

    (* ====== Logical Devices ====== *)
    (* Available LDs: AnUn_ArcProtInput1, Application, BinIO, BinIO_BinaryInputs, BinIO_BinaryOutputs, CB1, CB1_25Synchronization, CB1_Fundamental, Ds1, Ds2, Mod1, Mod1_Channel1, Mod2, Mod2_Channel1, Mod3, Mod3_Channel1, PowS, PowS_MeasPointI3ph1, PowS_MeasPointV1ph1, PowS_MeasPointV3ph1, Rec, Rec_FaultRecorder, VI1p1, VI1p1_Fundamental, VI3p1, VI3p1_5051NOCgndB1, VI3p1_5051OC3phase1, VI3p1_67DirOC3phB1, VI3p1_67NDirOCgndB1, VI3p1_ArcProtection1, VI3p1_Energy, VI3p1_FundSymComp, VI3p1_OperationalValues, VI3p1_ProcessMonitor, VI3p1_ExternalTrip1, VI3p1_ExternalTrip2, ComSupervision, ComSupervision_GOOSE *)

    (* ====== User Variables ====== *)
    (* Add your custom variables here *)
    (* Example:
    timer1: TON;
    counter: INT := 0;
    status_word: WORD;
    *)

END_VAR

(* ======================================================================
   INITIALIZATION SECTION
   Runs once on first scan. Use for setup and initialization.
   ====================================================================== *)
IF first_scan THEN
    (* Initialize user variables here *)
    cycle_count := 0;

    (* Log program start *)
    (* SCADA_LOG('INFO', CONCAT('PLC Program started: ', device_name)); *)

    first_scan := FALSE;
END_IF;

(* ======================================================================
   MAIN CYCLIC EXECUTION
   This section runs continuously every scan cycle (default 100ms).
   ====================================================================== *)

(* Increment cycle counter *)
cycle_count := cycle_count + 1;

(* ====== USER LOGIC SECTION 1: Pre-Processing ====== *)
(* Add logic that should run before main processing *)
(* Example:
IF ied_connected THEN
    (* Read IED data points *)
    (* status_word := READ_IED_DATA(device_name, 'LD0/MMXU1$MX$TotW$mag'); *)
END_IF;
*)

(* ====== USER LOGIC SECTION 2: Main Processing ====== *)
(* Add your main control logic here *)
(* Example:
IF counter > 100 THEN
    counter := 0;
    (* Perform periodic action *)
END_IF;
counter := counter + 1;
*)

(* ====== USER LOGIC SECTION 3: Post-Processing ====== *)
(* Add logic for outputs, writes, and cleanup *)
(* Example:
IF ied_connected THEN
    (* Write control commands to IED *)
    (* WRITE_IED_CONTROL(device_name, 'LD0/CSWI1$CO$Pos', TRUE); *)
END_IF;
*)

(* ====== Built-in Functions Available ====== *)
(*
   READ_IED_DATA(device: STRING, ref: STRING): ANY
       - Read data from IED object reference
       - Example: READ_IED_DATA('MyIED', 'LD0/MMXU1$MX$TotW$mag')

   WRITE_IED_DATA(device: STRING, ref: STRING, value: ANY): BOOL
       - Write data to IED object reference
       - Returns TRUE on success

   WRITE_IED_CONTROL(device: STRING, ref: STRING, value: ANY): BOOL
       - Send control command to IED
       - Returns TRUE on success

   SCADA_LOG(level: STRING, message: STRING)
       - Log message to event log
       - Levels: 'INFO', 'WARNING', 'ERROR'

   GET_DEVICE_STATUS(device: STRING): BOOL
       - Check if device is connected
*)

END_PROGRAM

(* ---- PRG_GPS03GCB08.st ---- *)
(* ========================================================================
   PLC PROGRAM: PRG_GPS03GCB08
   IED: GPS03GCB08
   Device: GPS03GCB08
   Generated: 2026-02-05 10:53:17

   This program runs cyclically (default 100ms) and has access to all
   data points of the associated IEC 61850 device. Users can add custom
   logic in the designated sections below.
   ======================================================================== *)

PROGRAM PRG_GPS03GCB08
VAR
    (* ====== System Variables ====== *)
    cycle_count: UDINT := 0;           (* Increments each scan cycle *)
    first_scan: BOOL := TRUE;          (* TRUE only on first execution *)
    scan_time_ms: REAL := 0.0;         (* Last scan time in milliseconds *)

    (* ====== IED Connection Status ====== *)
    ied_connected: BOOL := FALSE;      (* TRUE when IED server is running *)
    ied_name: STRING := 'GPS03GCB08';
    device_name: STRING := 'GPS03GCB08';

    (* ====== Logical Devices ====== *)
    (* Available LDs: AnUn_ArcProtInput1, Application, BinIO, BinIO_BinaryInputs, BinIO_BinaryOutputs, CB1, CB1_25Synchronization, CB1_Fundamental, Ds1, Ds2, Mod1, Mod1_Channel1, Mod2, Mod2_Channel1, Mod3, Mod3_Channel1, PowS, PowS_MeasPointI3ph1, PowS_MeasPointV1ph1, PowS_MeasPointV3ph1, Rec, Rec_FaultRecorder, VI1p1, VI1p1_Fundamental, VI3p1, VI3p1_5051NOCgndB1, VI3p1_5051OC3phase1, VI3p1_67DirOC3phB1, VI3p1_67NDirOCgndB1, VI3p1_ArcProtection1, VI3p1_Energy, VI3p1_FundSymComp, VI3p1_OperationalValues, VI3p1_ProcessMonitor, VI3p1_ExternalTrip1, VI3p1_ExternalTrip2, ComSupervision, ComSupervision_GOOSE *)

    (* ====== User Variables ====== *)
    (* Add your custom variables here *)
    (* Example:
    timer1: TON;
    counter: INT := 0;
    status_word: WORD;
    *)

END_VAR

(* ======================================================================
   INITIALIZATION SECTION
   Runs once on first scan. Use for setup and initialization.
   ====================================================================== *)
IF first_scan THEN
    (* Initialize user variables here *)
    cycle_count := 0;

    (* Log program start *)
    (* SCADA_LOG('INFO', CONCAT('PLC Program started: ', device_name)); *)

    first_scan := FALSE;
END_IF;

(* ======================================================================
   MAIN CYCLIC EXECUTION
   This section runs continuously every scan cycle (default 100ms).
   ====================================================================== *)

(* Increment cycle counter *)
cycle_count := cycle_count + 1;

(* ====== USER LOGIC SECTION 1: Pre-Processing ====== *)
(* Add logic that should run before main processing *)
(* Example:
IF ied_connected THEN
    (* Read IED data points *)
    (* status_word := READ_IED_DATA(device_name, 'LD0/MMXU1$MX$TotW$mag'); *)
END_IF;
*)

(* ====== USER LOGIC SECTION 2: Main Processing ====== *)
(* Add your main control logic here *)
(* Example:
IF counter > 100 THEN
    counter := 0;
    (* Perform periodic action *)
END_IF;
counter := counter + 1;
*)

(* ====== USER LOGIC SECTION 3: Post-Processing ====== *)
(* Add logic for outputs, writes, and cleanup *)
(* Example:
IF ied_connected THEN
    (* Write control commands to IED *)
    (* WRITE_IED_CONTROL(device_name, 'LD0/CSWI1$CO$Pos', TRUE); *)
END_IF;
*)

(* ====== Built-in Functions Available ====== *)
(*
   READ_IED_DATA(device: STRING, ref: STRING): ANY
       - Read data from IED object reference
       - Example: READ_IED_DATA('MyIED', 'LD0/MMXU1$MX$TotW$mag')

   WRITE_IED_DATA(device: STRING, ref: STRING, value: ANY): BOOL
       - Write data to IED object reference
       - Returns TRUE on success

   WRITE_IED_CONTROL(device: STRING, ref: STRING, value: ANY): BOOL
       - Send control command to IED
       - Returns TRUE on success

   SCADA_LOG(level: STRING, message: STRING)
       - Log message to event log
       - Levels: 'INFO', 'WARNING', 'ERROR'

   GET_DEVICE_STATUS(device: STRING): BOOL
       - Check if device is connected
*)

END_PROGRAM

(* ---- PRG_GPS03GCB09.st ---- *)
(* ========================================================================
   PLC PROGRAM: PRG_GPS03GCB09
   IED: GPS03GCB09
   Device: GPS03GCB09
   Generated: 2026-02-05 10:53:10

   This program runs cyclically (default 100ms) and has access to all
   data points of the associated IEC 61850 device. Users can add custom
   logic in the designated sections below.
   ======================================================================== *)

PROGRAM PRG_GPS03GCB09
VAR
    (* ====== System Variables ====== *)
    cycle_count: UDINT := 0;           (* Increments each scan cycle *)
    first_scan: BOOL := TRUE;          (* TRUE only on first execution *)
    scan_time_ms: REAL := 0.0;         (* Last scan time in milliseconds *)

    (* ====== IED Connection Status ====== *)
    ied_connected: BOOL := FALSE;      (* TRUE when IED server is running *)
    ied_name: STRING := 'GPS03GCB09';
    device_name: STRING := 'GPS03GCB09';

    (* ====== Logical Devices ====== *)
    (* Available LDs: AnUn_ArcProtInput1, Application, BinIO, BinIO_BinaryInputs, BinIO_BinaryOutputs, CB1, CB1_25Synchronization, CB1_Fundamental, Ds1, Ds2, Mod1, Mod1_Channel1, Mod2, Mod2_Channel1, Mod3, Mod3_Channel1, PowS, PowS_MeasPointI3ph1, PowS_MeasPointV1ph1, PowS_MeasPointV3ph1, Rec, Rec_FaultRecorder, VI1p1, VI1p1_Fundamental, VI3p1, VI3p1_5051NOCgndB1, VI3p1_5051OC3phase1, VI3p1_67DirOC3phB1, VI3p1_67NDirOCgndB1, VI3p1_ArcProtection1, VI3p1_Energy, VI3p1_FundSymComp, VI3p1_OperationalValues, VI3p1_ProcessMonitor, VI3p1_ExternalTrip1, VI3p1_ExternalTrip2, ComSupervision, ComSupervision_GOOSE *)

    (* ====== User Variables ====== *)
    (* Add your custom variables here *)
    (* Example:
    timer1: TON;
    counter: INT := 0;
    status_word: WORD;
    *)

END_VAR

(* ======================================================================
   INITIALIZATION SECTION
   Runs once on first scan. Use for setup and initialization.
   ====================================================================== *)
IF first_scan THEN
    (* Initialize user variables here *)
    cycle_count := 0;

    (* Log program start *)
    (* SCADA_LOG('INFO', CONCAT('PLC Program started: ', device_name)); *)

    first_scan := FALSE;
END_IF;

(* ======================================================================
   MAIN CYCLIC EXECUTION
   This section runs continuously every scan cycle (default 100ms).
   ====================================================================== *)

(* Increment cycle counter *)
cycle_count := cycle_count + 1;

(* ====== USER LOGIC SECTION 1: Pre-Processing ====== *)
(* Add logic that should run before main processing *)
(* Example:
IF ied_connected THEN
    (* Read IED data points *)
    (* status_word := READ_IED_DATA(device_name, 'LD0/MMXU1$MX$TotW$mag'); *)
END_IF;
*)

(* ====== USER LOGIC SECTION 2: Main Processing ====== *)
(* Add your main control logic here *)
(* Example:
IF counter > 100 THEN
    counter := 0;
    (* Perform periodic action *)
END_IF;
counter := counter + 1;
*)

(* ====== USER LOGIC SECTION 3: Post-Processing ====== *)
(* Add logic for outputs, writes, and cleanup *)
(* Example:
IF ied_connected THEN
    (* Write control commands to IED *)
    (* WRITE_IED_CONTROL(device_name, 'LD0/CSWI1$CO$Pos', TRUE); *)
END_IF;
*)

(* ====== Built-in Functions Available ====== *)
(*
   READ_IED_DATA(device: STRING, ref: STRING): ANY
       - Read data from IED object reference
       - Example: READ_IED_DATA('MyIED', 'LD0/MMXU1$MX$TotW$mag')

   WRITE_IED_DATA(device: STRING, ref: STRING, value: ANY): BOOL
       - Write data to IED object reference
       - Returns TRUE on success

   WRITE_IED_CONTROL(device: STRING, ref: STRING, value: ANY): BOOL
       - Send control command to IED
       - Returns TRUE on success

   SCADA_LOG(level: STRING, message: STRING)
       - Log message to event log
       - Levels: 'INFO', 'WARNING', 'ERROR'

   GET_DEVICE_STATUS(device: STRING): BOOL
       - Check if device is connected
*)

END_PROGRAM

(* ---- PRG_GPS03GCB10.st ---- *)
(* ========================================================================
   PLC PROGRAM: PRG_GPS03GCB10
   IED: GPS03GCB10
   Device: GPS03GCB10
   Generated: 2026-02-05 10:53:02

   This program runs cyclically (default 100ms) and has access to all
   data points of the associated IEC 61850 device. Users can add custom
   logic in the designated sections below.
   ======================================================================== *)

PROGRAM PRG_GPS03GCB10
VAR
    (* ====== System Variables ====== *)
    cycle_count: UDINT := 0;           (* Increments each scan cycle *)
    first_scan: BOOL := TRUE;          (* TRUE only on first execution *)
    scan_time_ms: REAL := 0.0;         (* Last scan time in milliseconds *)

    (* ====== IED Connection Status ====== *)
    ied_connected: BOOL := FALSE;      (* TRUE when IED server is running *)
    ied_name: STRING := 'GPS03GCB10';
    device_name: STRING := 'GPS03GCB10';

    (* ====== Logical Devices ====== *)
    (* Available LDs: AnUn_ArcProtInput1, Application, BinIO, BinIO_BinaryInputs, BinIO_BinaryOutputs, CB1, CB1_25Synchronization, CB1_Fundamental, Ds1, Ds2, Mod1, Mod1_Channel1, Mod2, Mod2_Channel1, Mod3, Mod3_Channel1, PowS, PowS_MeasPointI3ph1, PowS_MeasPointV1ph1, PowS_MeasPointV3ph1, Rec, Rec_FaultRecorder, VI1p1, VI1p1_Fundamental, VI3p1, VI3p1_5051NOCgndB1, VI3p1_5051OC3phase1, VI3p1_67DirOC3phB1, VI3p1_67NDirOCgndB1, VI3p1_ArcProtection1, VI3p1_Energy, VI3p1_FundSymComp, VI3p1_OperationalValues, VI3p1_ProcessMonitor, VI3p1_ExternalTrip1, VI3p1_ExternalTrip2, ComSupervision, ComSupervision_GOOSE *)

    (* ====== User Variables ====== *)
    (* Add your custom variables here *)
    (* Example:
    timer1: TON;
    counter: INT := 0;
    status_word: WORD;
    *)

END_VAR

(* ======================================================================
   INITIALIZATION SECTION
   Runs once on first scan. Use for setup and initialization.
   ====================================================================== *)
IF first_scan THEN
    (* Initialize user variables here *)
    cycle_count := 0;

    (* Log program start *)
    (* SCADA_LOG('INFO', CONCAT('PLC Program started: ', device_name)); *)

    first_scan := FALSE;
END_IF;

(* ======================================================================
   MAIN CYCLIC EXECUTION
   This section runs continuously every scan cycle (default 100ms).
   ====================================================================== *)

(* Increment cycle counter *)
cycle_count := cycle_count + 1;

(* ====== USER LOGIC SECTION 1: Pre-Processing ====== *)
(* Add logic that should run before main processing *)
(* Example:
IF ied_connected THEN
    (* Read IED data points *)
    (* status_word := READ_IED_DATA(device_name, 'LD0/MMXU1$MX$TotW$mag'); *)
END_IF;
*)

(* ====== USER LOGIC SECTION 2: Main Processing ====== *)
(* Add your main control logic here *)
(* Example:
IF counter > 100 THEN
    counter := 0;
    (* Perform periodic action *)
END_IF;
counter := counter + 1;
*)

(* ====== USER LOGIC SECTION 3: Post-Processing ====== *)
(* Add logic for outputs, writes, and cleanup *)
(* Example:
IF ied_connected THEN
    (* Write control commands to IED *)
    (* WRITE_IED_CONTROL(device_name, 'LD0/CSWI1$CO$Pos', TRUE); *)
END_IF;
*)

(* ====== Built-in Functions Available ====== *)
(*
   READ_IED_DATA(device: STRING, ref: STRING): ANY
       - Read data from IED object reference
       - Example: READ_IED_DATA('MyIED', 'LD0/MMXU1$MX$TotW$mag')

   WRITE_IED_DATA(device: STRING, ref: STRING, value: ANY): BOOL
       - Write data to IED object reference
       - Returns TRUE on success

   WRITE_IED_CONTROL(device: STRING, ref: STRING, value: ANY): BOOL
       - Send control command to IED
       - Returns TRUE on success

   SCADA_LOG(level: STRING, message: STRING)
       - Log message to event log
       - Levels: 'INFO', 'WARNING', 'ERROR'

   GET_DEVICE_STATUS(device: STRING): BOOL
       - Check if device is connected
*)

END_PROGRAM

(* ---- PRG_GPS03GCB11.st ---- *)
(* ========================================================================
   PLC PROGRAM: PRG_GPS03GCB11
   IED: GPS03GCB11
   Device: GPS03GCB11
   Generated: 2026-02-05 10:52:58

   This program runs cyclically (default 100ms) and has access to all
   data points of the associated IEC 61850 device. Users can add custom
   logic in the designated sections below.
   ======================================================================== *)

PROGRAM PRG_GPS03GCB11
VAR
    (* ====== System Variables ====== *)
    cycle_count: UDINT := 0;           (* Increments each scan cycle *)
    first_scan: BOOL := TRUE;          (* TRUE only on first execution *)
    scan_time_ms: REAL := 0.0;         (* Last scan time in milliseconds *)

    (* ====== IED Connection Status ====== *)
    ied_connected: BOOL := FALSE;      (* TRUE when IED server is running *)
    ied_name: STRING := 'GPS03GCB11';
    device_name: STRING := 'GPS03GCB11';

    (* ====== Logical Devices ====== *)
    (* Available LDs: AnUn_ArcProtInput1, Application, BinIO, BinIO_BinaryInputs, BinIO_BinaryOutputs, CB1, CB1_25Synchronization, CB1_Fundamental, Ds1, Ds2, Mod1, Mod1_Channel1, Mod2, Mod2_Channel1, Mod3, Mod3_Channel1, PowS, PowS_MeasPointI3ph1, PowS_MeasPointV1ph1, PowS_MeasPointV3ph1, Rec, Rec_FaultRecorder, VI1p1, VI1p1_Fundamental, VI3p1, VI3p1_5051NOCgndB1, VI3p1_5051OC3phase1, VI3p1_67DirOC3phB1, VI3p1_67NDirOCgndB1, VI3p1_ArcProtection1, VI3p1_Energy, VI3p1_FundSymComp, VI3p1_OperationalValues, VI3p1_ProcessMonitor, VI3p1_ExternalTrip1, VI3p1_ExternalTrip2, ComSupervision, ComSupervision_GOOSE *)

    (* ====== User Variables ====== *)
    (* Add your custom variables here *)
    (* Example:
    timer1: TON;
    counter: INT := 0;
    status_word: WORD;
    *)

END_VAR

(* ======================================================================
   INITIALIZATION SECTION
   Runs once on first scan. Use for setup and initialization.
   ====================================================================== *)
IF first_scan THEN
    (* Initialize user variables here *)
    cycle_count := 0;

    (* Log program start *)
    (* SCADA_LOG('INFO', CONCAT('PLC Program started: ', device_name)); *)

    first_scan := FALSE;
END_IF;

(* ======================================================================
   MAIN CYCLIC EXECUTION
   This section runs continuously every scan cycle (default 100ms).
   ====================================================================== *)

(* Increment cycle counter *)
cycle_count := cycle_count + 1;

(* ====== USER LOGIC SECTION 1: Pre-Processing ====== *)
(* Add logic that should run before main processing *)
(* Example:
IF ied_connected THEN
    (* Read IED data points *)
    (* status_word := READ_IED_DATA(device_name, 'LD0/MMXU1$MX$TotW$mag'); *)
END_IF;
*)

(* ====== USER LOGIC SECTION 2: Main Processing ====== *)
(* Add your main control logic here *)
(* Example:
IF counter > 100 THEN
    counter := 0;
    (* Perform periodic action *)
END_IF;
counter := counter + 1;
*)

(* ====== USER LOGIC SECTION 3: Post-Processing ====== *)
(* Add logic for outputs, writes, and cleanup *)
(* Example:
IF ied_connected THEN
    (* Write control commands to IED *)
    (* WRITE_IED_CONTROL(device_name, 'LD0/CSWI1$CO$Pos', TRUE); *)
END_IF;
*)

(* ====== Built-in Functions Available ====== *)
(*
   READ_IED_DATA(device: STRING, ref: STRING): ANY
       - Read data from IED object reference
       - Example: READ_IED_DATA('MyIED', 'LD0/MMXU1$MX$TotW$mag')

   WRITE_IED_DATA(device: STRING, ref: STRING, value: ANY): BOOL
       - Write data to IED object reference
       - Returns TRUE on success

   WRITE_IED_CONTROL(device: STRING, ref: STRING, value: ANY): BOOL
       - Send control command to IED
       - Returns TRUE on success

   SCADA_LOG(level: STRING, message: STRING)
       - Log message to event log
       - Levels: 'INFO', 'WARNING', 'ERROR'

   GET_DEVICE_STATUS(device: STRING): BOOL
       - Check if device is connected
*)

END_PROGRAM

(* ---- PRG_GPS03GCB12.st ---- *)
(* ========================================================================
   PLC PROGRAM: PRG_GPS03GCB12
   IED: GPS03GCB12
   Device: GPS03GCB12
   Generated: 2026-02-05 10:52:51

   This program runs cyclically (default 100ms) and has access to all
   data points of the associated IEC 61850 device. Users can add custom
   logic in the designated sections below.
   ======================================================================== *)

PROGRAM PRG_GPS03GCB12
VAR
    (* ====== System Variables ====== *)
    cycle_count: UDINT := 0;           (* Increments each scan cycle *)
    first_scan: BOOL := TRUE;          (* TRUE only on first execution *)
    scan_time_ms: REAL := 0.0;         (* Last scan time in milliseconds *)

    (* ====== IED Connection Status ====== *)
    ied_connected: BOOL := FALSE;      (* TRUE when IED server is running *)
    ied_name: STRING := 'GPS03GCB12';
    device_name: STRING := 'GPS03GCB12';

    (* ====== Logical Devices ====== *)
    (* Available LDs: AnUn_ArcProtInput1, Application, BinIO, BinIO_BinaryInputs, BinIO_BinaryOutputs, CB1, CB1_25Synchronization, CB1_Fundamental, Ds1, Ds2, Mod1, Mod1_Channel1, Mod2, Mod2_Channel1, Mod3, Mod3_Channel1, PowS, PowS_MeasPointI3ph1, PowS_MeasPointV1ph1, PowS_MeasPointV3ph1, Rec, Rec_FaultRecorder, VI1p1, VI1p1_Fundamental, VI3p1, VI3p1_5051NOCgndB1, VI3p1_5051OC3phase1, VI3p1_67DirOC3phB1, VI3p1_67NDirOCgndB1, VI3p1_ArcProtection1, VI3p1_Energy, VI3p1_FundSymComp, VI3p1_OperationalValues, VI3p1_ProcessMonitor, VI3p1_ExternalTrip1, VI3p1_ExternalTrip2, ComSupervision, ComSupervision_GOOSE *)

    (* ====== User Variables ====== *)
    (* Add your custom variables here *)
    (* Example:
    timer1: TON;
    counter: INT := 0;
    status_word: WORD;
    *)

END_VAR

(* ======================================================================
   INITIALIZATION SECTION
   Runs once on first scan. Use for setup and initialization.
   ====================================================================== *)
IF first_scan THEN
    (* Initialize user variables here *)
    cycle_count := 0;

    (* Log program start *)
    (* SCADA_LOG('INFO', CONCAT('PLC Program started: ', device_name)); *)

    first_scan := FALSE;
END_IF;

(* ======================================================================
   MAIN CYCLIC EXECUTION
   This section runs continuously every scan cycle (default 100ms).
   ====================================================================== *)

(* Increment cycle counter *)
cycle_count := cycle_count + 1;

(* ====== USER LOGIC SECTION 1: Pre-Processing ====== *)
(* Add logic that should run before main processing *)
(* Example:
IF ied_connected THEN
    (* Read IED data points *)
    (* status_word := READ_IED_DATA(device_name, 'LD0/MMXU1$MX$TotW$mag'); *)
END_IF;
*)

(* ====== USER LOGIC SECTION 2: Main Processing ====== *)
(* Add your main control logic here *)
(* Example:
IF counter > 100 THEN
    counter := 0;
    (* Perform periodic action *)
END_IF;
counter := counter + 1;
*)

(* ====== USER LOGIC SECTION 3: Post-Processing ====== *)
(* Add logic for outputs, writes, and cleanup *)
(* Example:
IF ied_connected THEN
    (* Write control commands to IED *)
    (* WRITE_IED_CONTROL(device_name, 'LD0/CSWI1$CO$Pos', TRUE); *)
END_IF;
*)

(* ====== Built-in Functions Available ====== *)
(*
   READ_IED_DATA(device: STRING, ref: STRING): ANY
       - Read data from IED object reference
       - Example: READ_IED_DATA('MyIED', 'LD0/MMXU1$MX$TotW$mag')

   WRITE_IED_DATA(device: STRING, ref: STRING, value: ANY): BOOL
       - Write data to IED object reference
       - Returns TRUE on success

   WRITE_IED_CONTROL(device: STRING, ref: STRING, value: ANY): BOOL
       - Send control command to IED
       - Returns TRUE on success

   SCADA_LOG(level: STRING, message: STRING)
       - Log message to event log
       - Levels: 'INFO', 'WARNING', 'ERROR'

   GET_DEVICE_STATUS(device: STRING): BOOL
       - Check if device is connected
*)

END_PROGRAM

(* ---- PRG_GPS03GPC01UPM01FCB01.st ---- *)
(* ========================================================================
   PLC PROGRAM: PRG_GPS03GPC01UPM01FCB01
   IED: GPS03GPC01UPM01FCB01
   Device: GPS03GPC01UPM01FCB01
   Generated: 2026-02-05 10:48:21

   This program runs cyclically (default 100ms) and has access to all
   data points of the associated IEC 61850 device. Users can add custom
   logic in the designated sections below.
   ======================================================================== *)

PROGRAM PRG_GPS03GPC01UPM01FCB01
VAR
    (* ====== System Variables ====== *)
    cycle_count: UDINT := 0;           (* Increments each scan cycle *)
    first_scan: BOOL := TRUE;          (* TRUE only on first execution *)
    scan_time_ms: REAL := 0.0;         (* Last scan time in milliseconds *)

    (* ====== IED Connection Status ====== *)
    ied_connected: BOOL := FALSE;      (* TRUE when IED server is running *)
    ied_name: STRING := 'GPS03GPC01UPM01FCB01';
    device_name: STRING := 'GPS03GPC01UPM01FCB01';

    (* ====== Logical Devices ====== *)
    (* Available LDs: AnUn_ArcProtInput1, Application, BinIO, BinIO_BinaryInputs, BinIO_BinaryOutputs, CB1, CB1_Fundamental, Ds1, Ds2, Mod1, Mod1_Channel1, Mod2, Mod2_Channel1, Mod3, Mod3_Channel1, PowS, PowS_MeasPointI3ph1, PowS_MeasPointV3ph1, Rec, Rec_FaultRecorder, VI3p1, VI3p1_5051NOCgndB1, VI3p1_5051OC3phase1, VI3p1_ArcProtection1, VI3p1_Energy, VI3p1_FundSymComp, VI3p1_OperationalValues, VI3p1_ProcessMonitor, VI3p1_ExternalTrip1, VI3p1_67DirOC3phB1, VI3p1_67NDirOCgndB1, ComSupervision, ComSupervision_GOOSE *)

    (* ====== User Variables ====== *)
    (* Add your custom variables here *)
    (* Example:
    timer1: TON;
    counter: INT := 0;
    status_word: WORD;
    *)

END_VAR

(* ======================================================================
   INITIALIZATION SECTION
   Runs once on first scan. Use for setup and initialization.
   ====================================================================== *)
IF first_scan THEN
    (* Initialize user variables here *)
    cycle_count := 0;

    (* Log program start *)
    (* SCADA_LOG('INFO', CONCAT('PLC Program started: ', device_name)); *)

    first_scan := FALSE;
END_IF;

(* ======================================================================
   MAIN CYCLIC EXECUTION
   This section runs continuously every scan cycle (default 100ms).
   ====================================================================== *)

(* Increment cycle counter *)
cycle_count := cycle_count + 1;

(* ====== USER LOGIC SECTION 1: Pre-Processing ====== *)
(* Add logic that should run before main processing *)
(* Example:
IF ied_connected THEN
    (* Read IED data points *)
    (* status_word := READ_IED_DATA(device_name, 'LD0/MMXU1$MX$TotW$mag'); *)
END_IF;
*)

(* ====== USER LOGIC SECTION 2: Main Processing ====== *)
(* Add your main control logic here *)
(* Example:
IF counter > 100 THEN
    counter := 0;
    (* Perform periodic action *)
END_IF;
counter := counter + 1;
*)

(* ====== USER LOGIC SECTION 3: Post-Processing ====== *)
(* Add logic for outputs, writes, and cleanup *)
(* Example:
IF ied_connected THEN
    (* Write control commands to IED *)
    (* WRITE_IED_CONTROL(device_name, 'LD0/CSWI1$CO$Pos', TRUE); *)
END_IF;
*)

(* ====== Built-in Functions Available ====== *)
(*
   READ_IED_DATA(device: STRING, ref: STRING): ANY
       - Read data from IED object reference
       - Example: READ_IED_DATA('MyIED', 'LD0/MMXU1$MX$TotW$mag')

   WRITE_IED_DATA(device: STRING, ref: STRING, value: ANY): BOOL
       - Write data to IED object reference
       - Returns TRUE on success

   WRITE_IED_CONTROL(device: STRING, ref: STRING, value: ANY): BOOL
       - Send control command to IED
       - Returns TRUE on success

   SCADA_LOG(level: STRING, message: STRING)
       - Log message to event log
       - Levels: 'INFO', 'WARNING', 'ERROR'

   GET_DEVICE_STATUS(device: STRING): BOOL
       - Check if device is connected
*)

END_PROGRAM

(* ---- PRG_GPS03GPC01UPM01FCB02.st ---- *)
(* ========================================================================
   PLC PROGRAM: PRG_GPS03GPC01UPM01FCB02
   IED: GPS03GPC01UPM01FCB02
   Device: GPS03GPC01UPM01FCB02
   Generated: 2026-02-05 10:48:27

   This program runs cyclically (default 100ms) and has access to all
   data points of the associated IEC 61850 device. Users can add custom
   logic in the designated sections below.
   ======================================================================== *)

PROGRAM PRG_GPS03GPC01UPM01FCB02
VAR
    (* ====== System Variables ====== *)
    cycle_count: UDINT := 0;           (* Increments each scan cycle *)
    first_scan: BOOL := TRUE;          (* TRUE only on first execution *)
    scan_time_ms: REAL := 0.0;         (* Last scan time in milliseconds *)

    (* ====== IED Connection Status ====== *)
    ied_connected: BOOL := FALSE;      (* TRUE when IED server is running *)
    ied_name: STRING := 'GPS03GPC01UPM01FCB02';
    device_name: STRING := 'GPS03GPC01UPM01FCB02';

    (* ====== Logical Devices ====== *)
    (* Available LDs: AnUn_ArcProtInput1, Application, BinIO, BinIO_BinaryInputs, BinIO_BinaryOutputs, CB1, CB1_Fundamental, Ds1, Ds2, Mod1, Mod1_Channel1, Mod2, Mod2_Channel1, Mod3, Mod3_Channel1, PowS, PowS_MeasPointI3ph1, PowS_MeasPointV3ph1, Rec, Rec_FaultRecorder, VI3p1, VI3p1_5051NOCgndB1, VI3p1_5051OC3phase1, VI3p1_ArcProtection1, VI3p1_Energy, VI3p1_FundSymComp, VI3p1_OperationalValues, VI3p1_ProcessMonitor, VI3p1_ExternalTrip1, VI3p1_67DirOC3phB1, VI3p1_67NDirOCgndB1, ComSupervision, ComSupervision_GOOSE *)

    (* ====== User Variables ====== *)
    (* Add your custom variables here *)
    (* Example:
    timer1: TON;
    counter: INT := 0;
    status_word: WORD;
    *)

END_VAR

(* ======================================================================
   INITIALIZATION SECTION
   Runs once on first scan. Use for setup and initialization.
   ====================================================================== *)
IF first_scan THEN
    (* Initialize user variables here *)
    cycle_count := 0;

    (* Log program start *)
    (* SCADA_LOG('INFO', CONCAT('PLC Program started: ', device_name)); *)

    first_scan := FALSE;
END_IF;

(* ======================================================================
   MAIN CYCLIC EXECUTION
   This section runs continuously every scan cycle (default 100ms).
   ====================================================================== *)

(* Increment cycle counter *)
cycle_count := cycle_count + 1;

(* ====== USER LOGIC SECTION 1: Pre-Processing ====== *)
(* Add logic that should run before main processing *)
(* Example:
IF ied_connected THEN
    (* Read IED data points *)
    (* status_word := READ_IED_DATA(device_name, 'LD0/MMXU1$MX$TotW$mag'); *)
END_IF;
*)

(* ====== USER LOGIC SECTION 2: Main Processing ====== *)
(* Add your main control logic here *)
(* Example:
IF counter > 100 THEN
    counter := 0;
    (* Perform periodic action *)
END_IF;
counter := counter + 1;
*)

(* ====== USER LOGIC SECTION 3: Post-Processing ====== *)
(* Add logic for outputs, writes, and cleanup *)
(* Example:
IF ied_connected THEN
    (* Write control commands to IED *)
    (* WRITE_IED_CONTROL(device_name, 'LD0/CSWI1$CO$Pos', TRUE); *)
END_IF;
*)

(* ====== Built-in Functions Available ====== *)
(*
   READ_IED_DATA(device: STRING, ref: STRING): ANY
       - Read data from IED object reference
       - Example: READ_IED_DATA('MyIED', 'LD0/MMXU1$MX$TotW$mag')

   WRITE_IED_DATA(device: STRING, ref: STRING, value: ANY): BOOL
       - Write data to IED object reference
       - Returns TRUE on success

   WRITE_IED_CONTROL(device: STRING, ref: STRING, value: ANY): BOOL
       - Send control command to IED
       - Returns TRUE on success

   SCADA_LOG(level: STRING, message: STRING)
       - Log message to event log
       - Levels: 'INFO', 'WARNING', 'ERROR'

   GET_DEVICE_STATUS(device: STRING): BOOL
       - Check if device is connected
*)

END_PROGRAM

(* ---- PRG_GPS03GPC01UPM01MCB01.st ---- *)
(* ========================================================================
   PLC PROGRAM: PRG_GPS03GPC01UPM01MCB01
   IED: GPS03GPC01UPM01MCB01
   Device: GPS03GPC01UPM01MCB01
   Generated: 2026-02-05 10:48:29

   This program runs cyclically (default 100ms) and has access to all
   data points of the associated IEC 61850 device. Users can add custom
   logic in the designated sections below.
   ======================================================================== *)

PROGRAM PRG_GPS03GPC01UPM01MCB01
VAR
    (* ====== System Variables ====== *)
    cycle_count: UDINT := 0;           (* Increments each scan cycle *)
    first_scan: BOOL := TRUE;          (* TRUE only on first execution *)
    scan_time_ms: REAL := 0.0;         (* Last scan time in milliseconds *)

    (* ====== IED Connection Status ====== *)
    ied_connected: BOOL := FALSE;      (* TRUE when IED server is running *)
    ied_name: STRING := 'GPS03GPC01UPM01MCB01';
    device_name: STRING := 'GPS03GPC01UPM01MCB01';

    (* ====== Logical Devices ====== *)
    (* Available LDs: AnUn_ArcProtInput1, Application, BinIO, BinIO_BinaryInputs, BinIO_BinaryOutputs, CB1, CB1_Fundamental, Ds1, Ds2, Mod1, Mod1_Channel1, Mod2, Mod2_Channel1, Mod3, Mod3_Channel1, PowS, PowS_MeasPointI3ph1, PowS_MeasPointV3ph1, Rec, Rec_FaultRecorder, VI3p1, VI3p1_5051NOCgndB1, VI3p1_5051OC3phase1, VI3p1_ArcProtection1, VI3p1_Energy, VI3p1_FundSymComp, VI3p1_OperationalValues, VI3p1_ProcessMonitor, VI3p1_ExternalTrip1, VI3p1_67DirOC3phB1, VI3p1_67NDirOCgndB1, VI3p1_ExternalTrip2, ComSupervision, ComSupervision_GOOSE *)

    (* ====== User Variables ====== *)
    (* Add your custom variables here *)
    (* Example:
    timer1: TON;
    counter: INT := 0;
    status_word: WORD;
    *)

END_VAR

(* ======================================================================
   INITIALIZATION SECTION
   Runs once on first scan. Use for setup and initialization.
   ====================================================================== *)
IF first_scan THEN
    (* Initialize user variables here *)
    cycle_count := 0;

    (* Log program start *)
    (* SCADA_LOG('INFO', CONCAT('PLC Program started: ', device_name)); *)

    first_scan := FALSE;
END_IF;

(* ======================================================================
   MAIN CYCLIC EXECUTION
   This section runs continuously every scan cycle (default 100ms).
   ====================================================================== *)

(* Increment cycle counter *)
cycle_count := cycle_count + 1;

(* ====== USER LOGIC SECTION 1: Pre-Processing ====== *)
(* Add logic that should run before main processing *)
(* Example:
IF ied_connected THEN
    (* Read IED data points *)
    (* status_word := READ_IED_DATA(device_name, 'LD0/MMXU1$MX$TotW$mag'); *)
END_IF;
*)

(* ====== USER LOGIC SECTION 2: Main Processing ====== *)
(* Add your main control logic here *)
(* Example:
IF counter > 100 THEN
    counter := 0;
    (* Perform periodic action *)
END_IF;
counter := counter + 1;
*)

(* ====== USER LOGIC SECTION 3: Post-Processing ====== *)
(* Add logic for outputs, writes, and cleanup *)
(* Example:
IF ied_connected THEN
    (* Write control commands to IED *)
    (* WRITE_IED_CONTROL(device_name, 'LD0/CSWI1$CO$Pos', TRUE); *)
END_IF;
*)

(* ====== Built-in Functions Available ====== *)
(*
   READ_IED_DATA(device: STRING, ref: STRING): ANY
       - Read data from IED object reference
       - Example: READ_IED_DATA('MyIED', 'LD0/MMXU1$MX$TotW$mag')

   WRITE_IED_DATA(device: STRING, ref: STRING, value: ANY): BOOL
       - Write data to IED object reference
       - Returns TRUE on success

   WRITE_IED_CONTROL(device: STRING, ref: STRING, value: ANY): BOOL
       - Send control command to IED
       - Returns TRUE on success

   SCADA_LOG(level: STRING, message: STRING)
       - Log message to event log
       - Levels: 'INFO', 'WARNING', 'ERROR'

   GET_DEVICE_STATUS(device: STRING): BOOL
       - Check if device is connected
*)

END_PROGRAM

(* ---- PRG_GPS03GPC02UPM01FCB01.st ---- *)
(* ========================================================================
   PLC PROGRAM: PRG_GPS03GPC02UPM01FCB01
   IED: GPS03GPC02UPM01FCB01
   Device: GPS03GPC02UPM01FCB01
   Generated: 2026-02-05 10:48:32

   This program runs cyclically (default 100ms) and has access to all
   data points of the associated IEC 61850 device. Users can add custom
   logic in the designated sections below.
   ======================================================================== *)

PROGRAM PRG_GPS03GPC02UPM01FCB01
VAR
    (* ====== System Variables ====== *)
    cycle_count: UDINT := 0;           (* Increments each scan cycle *)
    first_scan: BOOL := TRUE;          (* TRUE only on first execution *)
    scan_time_ms: REAL := 0.0;         (* Last scan time in milliseconds *)

    (* ====== IED Connection Status ====== *)
    ied_connected: BOOL := FALSE;      (* TRUE when IED server is running *)
    ied_name: STRING := 'GPS03GPC02UPM01FCB01';
    device_name: STRING := 'GPS03GPC02UPM01FCB01';

    (* ====== Logical Devices ====== *)
    (* Available LDs: AnUn_ArcProtInput1, Application, BinIO, BinIO_BinaryInputs, BinIO_BinaryOutputs, CB1, CB1_Fundamental, Ds1, Ds2, Mod1, Mod1_Channel1, Mod2, Mod2_Channel1, Mod3, Mod3_Channel1, PowS, PowS_MeasPointI3ph1, PowS_MeasPointV3ph1, Rec, Rec_FaultRecorder, VI3p1, VI3p1_5051NOCgndB1, VI3p1_5051OC3phase1, VI3p1_ArcProtection1, VI3p1_Energy, VI3p1_FundSymComp, VI3p1_OperationalValues, VI3p1_ProcessMonitor, VI3p1_ExternalTrip1, VI3p1_67DirOC3phB1, VI3p1_67NDirOCgndB1, ComSupervision, ComSupervision_GOOSE *)

    (* ====== User Variables ====== *)
    (* Add your custom variables here *)
    (* Example:
    timer1: TON;
    counter: INT := 0;
    status_word: WORD;
    *)

END_VAR

(* ======================================================================
   INITIALIZATION SECTION
   Runs once on first scan. Use for setup and initialization.
   ====================================================================== *)
IF first_scan THEN
    (* Initialize user variables here *)
    cycle_count := 0;

    (* Log program start *)
    (* SCADA_LOG('INFO', CONCAT('PLC Program started: ', device_name)); *)

    first_scan := FALSE;
END_IF;

(* ======================================================================
   MAIN CYCLIC EXECUTION
   This section runs continuously every scan cycle (default 100ms).
   ====================================================================== *)

(* Increment cycle counter *)
cycle_count := cycle_count + 1;

(* ====== USER LOGIC SECTION 1: Pre-Processing ====== *)
(* Add logic that should run before main processing *)
(* Example:
IF ied_connected THEN
    (* Read IED data points *)
    (* status_word := READ_IED_DATA(device_name, 'LD0/MMXU1$MX$TotW$mag'); *)
END_IF;
*)

(* ====== USER LOGIC SECTION 2: Main Processing ====== *)
(* Add your main control logic here *)
(* Example:
IF counter > 100 THEN
    counter := 0;
    (* Perform periodic action *)
END_IF;
counter := counter + 1;
*)

(* ====== USER LOGIC SECTION 3: Post-Processing ====== *)
(* Add logic for outputs, writes, and cleanup *)
(* Example:
IF ied_connected THEN
    (* Write control commands to IED *)
    (* WRITE_IED_CONTROL(device_name, 'LD0/CSWI1$CO$Pos', TRUE); *)
END_IF;
*)

(* ====== Built-in Functions Available ====== *)
(*
   READ_IED_DATA(device: STRING, ref: STRING): ANY
       - Read data from IED object reference
       - Example: READ_IED_DATA('MyIED', 'LD0/MMXU1$MX$TotW$mag')

   WRITE_IED_DATA(device: STRING, ref: STRING, value: ANY): BOOL
       - Write data to IED object reference
       - Returns TRUE on success

   WRITE_IED_CONTROL(device: STRING, ref: STRING, value: ANY): BOOL
       - Send control command to IED
       - Returns TRUE on success

   SCADA_LOG(level: STRING, message: STRING)
       - Log message to event log
       - Levels: 'INFO', 'WARNING', 'ERROR'

   GET_DEVICE_STATUS(device: STRING): BOOL
       - Check if device is connected
*)

END_PROGRAM

(* ---- PRG_GPS03GPC02UPM01FCB02.st ---- *)
(* ========================================================================
   PLC PROGRAM: PRG_GPS03GPC02UPM01FCB02
   IED: GPS03GPC02UPM01FCB02
   Device: GPS03GPC02UPM01FCB02
   Generated: 2026-02-05 10:48:41

   This program runs cyclically (default 100ms) and has access to all
   data points of the associated IEC 61850 device. Users can add custom
   logic in the designated sections below.
   ======================================================================== *)

PROGRAM PRG_GPS03GPC02UPM01FCB02
VAR
    (* ====== System Variables ====== *)
    cycle_count: UDINT := 0;           (* Increments each scan cycle *)
    first_scan: BOOL := TRUE;          (* TRUE only on first execution *)
    scan_time_ms: REAL := 0.0;         (* Last scan time in milliseconds *)

    (* ====== IED Connection Status ====== *)
    ied_connected: BOOL := FALSE;      (* TRUE when IED server is running *)
    ied_name: STRING := 'GPS03GPC02UPM01FCB02';
    device_name: STRING := 'GPS03GPC02UPM01FCB02';

    (* ====== Logical Devices ====== *)
    (* Available LDs: AnUn_ArcProtInput1, Application, BinIO, BinIO_BinaryInputs, BinIO_BinaryOutputs, CB1, CB1_Fundamental, Ds1, Ds2, Mod1, Mod1_Channel1, Mod2, Mod2_Channel1, Mod3, Mod3_Channel1, PowS, PowS_MeasPointI3ph1, PowS_MeasPointV3ph1, Rec, Rec_FaultRecorder, VI3p1, VI3p1_5051NOCgndB1, VI3p1_5051OC3phase1, VI3p1_ArcProtection1, VI3p1_Energy, VI3p1_FundSymComp, VI3p1_OperationalValues, VI3p1_ProcessMonitor, VI3p1_ExternalTrip1, VI3p1_67DirOC3phB1, VI3p1_67NDirOCgndB1, ComSupervision, ComSupervision_GOOSE *)

    (* ====== User Variables ====== *)
    (* Add your custom variables here *)
    (* Example:
    timer1: TON;
    counter: INT := 0;
    status_word: WORD;
    *)

END_VAR

(* ======================================================================
   INITIALIZATION SECTION
   Runs once on first scan. Use for setup and initialization.
   ====================================================================== *)
IF first_scan THEN
    (* Initialize user variables here *)
    cycle_count := 0;

    (* Log program start *)
    (* SCADA_LOG('INFO', CONCAT('PLC Program started: ', device_name)); *)

    first_scan := FALSE;
END_IF;

(* ======================================================================
   MAIN CYCLIC EXECUTION
   This section runs continuously every scan cycle (default 100ms).
   ====================================================================== *)

(* Increment cycle counter *)
cycle_count := cycle_count + 1;

(* ====== USER LOGIC SECTION 1: Pre-Processing ====== *)
(* Add logic that should run before main processing *)
(* Example:
IF ied_connected THEN
    (* Read IED data points *)
    (* status_word := READ_IED_DATA(device_name, 'LD0/MMXU1$MX$TotW$mag'); *)
END_IF;
*)

(* ====== USER LOGIC SECTION 2: Main Processing ====== *)
(* Add your main control logic here *)
(* Example:
IF counter > 100 THEN
    counter := 0;
    (* Perform periodic action *)
END_IF;
counter := counter + 1;
*)

(* ====== USER LOGIC SECTION 3: Post-Processing ====== *)
(* Add logic for outputs, writes, and cleanup *)
(* Example:
IF ied_connected THEN
    (* Write control commands to IED *)
    (* WRITE_IED_CONTROL(device_name, 'LD0/CSWI1$CO$Pos', TRUE); *)
END_IF;
*)

(* ====== Built-in Functions Available ====== *)
(*
   READ_IED_DATA(device: STRING, ref: STRING): ANY
       - Read data from IED object reference
       - Example: READ_IED_DATA('MyIED', 'LD0/MMXU1$MX$TotW$mag')

   WRITE_IED_DATA(device: STRING, ref: STRING, value: ANY): BOOL
       - Write data to IED object reference
       - Returns TRUE on success

   WRITE_IED_CONTROL(device: STRING, ref: STRING, value: ANY): BOOL
       - Send control command to IED
       - Returns TRUE on success

   SCADA_LOG(level: STRING, message: STRING)
       - Log message to event log
       - Levels: 'INFO', 'WARNING', 'ERROR'

   GET_DEVICE_STATUS(device: STRING): BOOL
       - Check if device is connected
*)

END_PROGRAM
